// Mitsubishi GX Works2 project: BookEX6_54 Socket   PLC: Q13UDV

// global labels: Global
VAR_GLOBAL
  bVar0 AT M5000 : BOOL;
  abArray0 AT M5010 : ARRAY [0..49] OF BOOL;
  sStr0 AT D5000 : STRING[199];
  sStr1 AT D5100 : STRING[199];
  sStr2 AT D5200 : STRING[199];
  sStr3 AT D5300 : STRING[199];
  sStr4 AT D5400 : STRING[199];
  sStr5 AT D5500 : STRING[199];
  sStr6 AT D5600 : STRING[199];
  sStr7 AT D5700 : STRING[199];
  sStr8 AT D5800 : STRING[199];
  sStr9 AT D5900 : STRING[199];
  iVar0 AT D4500 : INT;
  iVar1 AT D4501 : INT;
  iVar2 AT D4502 : INT;
  iVar3 AT D4503 : INT;
  iVar4 AT D4504 : INT;
  iVar5 AT D4505 : INT;
  iVar6 AT D4506 : INT;
  iVar7 AT D4507 : INT;
  iVar8 AT D4508 : INT;
  iVar9 AT D4509 : INT;
  dVar0 AT D4510 : DINT;
  dVar1 AT D4512 : DINT;
  dVar2 AT D4514 : DINT;
  dVar3 AT D4516 : DINT;
  dVar4 AT D4518 : DINT;
  dVar5 AT D4520 : DINT;
  dVar6 AT D4522 : DINT;
  dVar7 AT D4524 : DINT;
  dVar8 AT D4526 : DINT;
  dVar9 AT D4528 : DINT;
  wVar0 AT D4530 : WORD;
  wVar1 AT D4531 : WORD;
  wVar2 AT D4532 : WORD;
  wVar3 AT D4533 : WORD;
  wVar4 AT D4534 : WORD;
  wVar5 AT D4535 : WORD;
  wVar6 AT D4536 : WORD;
  wVar7 AT D4537 : WORD;
  wVar8 AT D4538 : WORD;
  wVar9 AT D4539 : WORD;
  dwVar0 AT D4540 : DWORD;
  dwVar1 AT D4542 : DWORD;
  dwVar2 AT D4544 : DWORD;
  dwVar3 AT D4546 : DWORD;
  dwVar4 AT D4548 : DWORD;
  dwVar5 AT D4550 : DWORD;
  dwVar6 AT D4552 : DWORD;
  dwVar7 AT D4554 : DWORD;
  dwVar8 AT D4556 : DWORD;
  dwVar9 AT D4558 : DWORD;
  fsVar0 AT D4560 : REAL;
  fsVar1 AT D4562 : REAL;
  fsVar2 AT D4564 : REAL;
  fsVar3 AT D4566 : REAL;
  fsVar4 AT D4568 : REAL;
  fsVar5 AT D4570 : REAL;
  fsVar6 AT D4572 : REAL;
  fsVar7 AT D4574 : REAL;
  fsVar8 AT D4576 : REAL;
  fsVar9 AT D4578 : REAL;
  fdVar0 AT D4580 : LREAL;
  tTime0 AT D4620 : TIME;
  tTime1 AT D4622 : TIME;
  tTime2 AT D4624 : TIME;
  tTime3 AT D4626 : TIME;
  tTime4 AT D4628 : TIME;
  tTime5 AT D4630 : TIME;
  tTime6 AT D4632 : TIME;
  tTime7 AT D4634 : TIME;
  tTime8 AT D4636 : TIME;
  tTime9 AT D4638 : TIME;
  tTime10 AT D4640 : TIME;
  bVar1 AT M5001 : BOOL;
  bVar2 AT M5002 : BOOL;
  bVar3 AT M5003 : BOOL;
  bVar4 AT M5004 : BOOL;
  bVar5 AT M5005 : BOOL;
  bVar6 AT M5006 : BOOL;
  bVar7 AT M5007 : BOOL;
  bVar8 AT M5008 : BOOL;
  bVar9 AT M5009 : BOOL;
  abArray1 AT M5060 : ARRAY [0..49] OF BOOL;
  abArray2 AT M5110 : ARRAY [0..49] OF BOOL;
  abArray3 AT M5160 : ARRAY [0..49] OF BOOL;
  abArray4 AT M5210 : ARRAY [0..49] OF BOOL;
  abArray5 AT M5260 : ARRAY [0..49] OF BOOL;
  abArray6 AT M5310 : ARRAY [0..49] OF BOOL;
  abArray7 AT M5360 : ARRAY [0..49] OF BOOL;
  abArray8 AT M5410 : ARRAY [0..49] OF BOOL;
  abArray9 AT M5460 : ARRAY [0..49] OF BOOL;
  fdVar1 AT D4584 : LREAL;
  fdVar2 AT D4588 : LREAL;
  fdVar3 AT D4592 : LREAL;
  fdVar4 AT D4596 : LREAL;
  fdVar5 AT D4600 : LREAL;
  fdVar6 AT D4604 : LREAL;
  fdVar7 AT D4608 : LREAL;
  fdVar8 AT D4612 : LREAL;
  fdVar9 AT D4616 : LREAL;
END_VAR

// global labels: QPLCSpecial
VAR_GLOBAL
  sbGetTime AT SM213 : BOOL;
  sbOn AT SM400 : BOOL;
  sbOff AT SM401 : BOOL;
  sbOn1Time AT SM402 : BOOL;
  sbOff1Time AT SM403 : BOOL;
  sb5ms AT SM409 : BOOL;
  sdSwitch AT SD200 : INT;
  sdTime03 AT SD212 : INT;
  sdTime04 AT SD213 : INT;
  sdTime02 AT SD211 : INT;
  sdTime01 AT SD210 : INT;
  sdScanTime1 AT SD521 : INT;
  sdScanTimeMin1 AT SD525 : INT;
  sdScanTimeMin AT SD524 : INT;
  sdScanTimeMax1 AT SD527 : INT;
  sdScanTimeMax AT SD526 : INT;
  sbErrInfo2 AT SM16 : BOOL;
  sbErrInfo AT SM5 : BOOL;
  sbSelfError AT SM1 : BOOL;
  sbDiagError AT SM0 : BOOL;
  sbResetErr AT SM50 : BOOL;
  sbSetTime AT SM210 : BOOL;
  sbFuse AT SM60 : BOOL;
  sbOpError AT SM56 : BOOL;
  sbPowerDown AT SM53 : BOOL;
  sbBatLow AT SM52 : BOOL;
  sbBatLowL AT SM51 : BOOL;
  sbSTOP AT SM203 : BOOL;
  sbPAUSE AT SM204 : BOOL;
  sbNsec AT SM414 : BOOL;
  sb1000ms AT SM413 : BOOL;
  sb500ms AT SM412 : BOOL;
  sbNms AT SM415 : BOOL;
  sbUserClk4 AT SM424 : BOOL;
  sbUserClk3 AT SM423 : BOOL;
  sbUserClk2 AT SM422 : BOOL;
  sbUserClk1 AT SM421 : BOOL;
  sbUserClk0 AT SM420 : BOOL;
  sdBatLowL AT SD51 : INT;
  sdPLCErrInfo AT SD4 : INT;
  sdPLCErrDate2 AT SD3 : INT;
  sdPLCErrDate1 AT SD2 : INT;
  sdPLCErrDate0 AT SD1 : INT;
  sdPLCErrCode AT SD0 : INT;
  sdFuse AT SD60 : INT;
  sdPowerDown AT SD53 : INT;
  sdBatLow AT SD52 : INT;
  sdCPUSts AT SD203 : INT;
  sdLed AT SD201 : INT;
  sdScanTime AT SD520 : INT;
  sdCntNsec AT SD414 : INT;
  sdCnt1sec AT SD412 : INT;
  sdCntScan AT SD420 : INT;
  sdCntNms AT SD415 : INT;
  sb100ms AT SM411 : BOOL;
  sb50ms AT SM410 : BOOL;
  sdSckOpenComp AT SD1282 : WORD;
  sdSckOpenReq AT SD1284 : WORD;
  sdSckDataRx AT SD1286 : WORD;
  sdSckConn AT SD1288 : WORD;
END_VAR

// global labels: Network
VAR_GLOBAL
  aSendData1 AT D100 : ARRAY [0..4] OF INT;
  aiTxData AT D4000 : ARRAY [0..99] OF INT;
  aiRxData AT D4100 : ARRAY [0..99] OF INT;
  iOpenOK AT D3900 : INT;
  iOpenERR AT D3901 : INT;
  iSendOK AT D3902 : INT;
  iSendERR AT D3903 : INT;
  iCloseOK AT D3906 : INT;
  iCloseERR AT D3907 : INT;
  iRecvOK AT D3904 : INT;
  iRecvERR AT D3905 : INT;
  aiTxData2 AT D4200 : ARRAY [0..99] OF INT;
  aiRxData2 AT D4300 : ARRAY [0..99] OF INT;
  iOpenOK2 AT D3908 : INT;
  iOpenERR2 AT D3909 : INT;
  iSendOK2 AT D3910 : INT;
  iSendERR2 AT D3911 : INT;
  iRecvOK2 AT D3912 : INT;
  iRecvERR2 AT D3913 : INT;
  iCloseOK2 AT D3914 : INT;
  iCloseERR2 AT D3915 : INT;
  iEOpenComp AT D3916 : INT;
  iEOpenReq AT D3917 : INT;
  iERecvFlag AT D3918 : INT;
  iOpenCode AT D3919 : INT;
  iSendCode AT D3920 : INT;
  iRecvCode AT D3921 : INT;
  iCloseCode AT D3922 : INT;
  iOpenCode2 AT D3923 : INT;
  iSendCode2 AT D3924 : INT;
  iRecvCode2 AT D3925 : INT;
  iCloseCode2 AT D3926 : INT;
  aRecvData1 AT D105 : ARRAY [0..4] OF INT;
  aSendData2 AT D110 : ARRAY [0..4] OF INT;
  aRecvData2 AT D115 : ARRAY [0..4] OF INT;
  aSendData3 AT D120 : ARRAY [0..4] OF INT;
  aRecvData3 AT D125 : ARRAY [0..4] OF INT;
  aRdata AT D140 : ARRAY [0..9] OF INT;
  aSLMPDataTx AT D150 : ARRAY [0..9] OF WORD;
  aSLMPDataRx AT D160 : ARRAY [0..9] OF WORD;
END_VAR
// user libraries (not included): HMI

PROGRAM Ex_CactEpas
VAR
  bOpenReqC : BOOL;
  bOpenOkC : BOOL;
  bOpenErrC : BOOL;
  abOpenResC : ARRAY [0..1] OF BOOL;
  acOpenData : ARRAY [0..9] OF INT;
  bSendReqC : BOOL;
  bSendOkC : BOOL;
  bSendErrC : BOOL;
  abSendResC : ARRAY [0..1] OF BOOL;
  acSendDataC : ARRAY [0..1] OF INT;
  bRecvOkC : BOOL;
  bRecvErrC : BOOL;
  abRecvResC : ARRAY [0..1] OF BOOL;
  bCloseReq : BOOL;
  bCloseOkC : BOOL;
  bCloseErrC : BOOL;
  abCloseResC : ARRAY [0..1] OF BOOL;
  acCloseData : ARRAY [0..1] OF INT;
  CntSend1 : INT;
  CntSend2 : INT;
  CntRecv1 : INT;
  CntRecv2 : INT;
  Mov4INT_1 : Mov4INT;
  Mov8INT_1 : Mov8INT;
  acRdCtrl : ARRAY [0..9] OF INT;
  Mov4INT_2 : Mov4INT;
  bOpenReqE : BOOL;
  bOpenOkE : BOOL;
  bOpenErrE : BOOL;
  abOpenResE : ARRAY [0..1] OF BOOL;
  bSendErrE : BOOL;
  bSendOkE : BOOL;
  bSendReqE : BOOL;
  abSendResE : ARRAY [0..1] OF BOOL;
  abRecvResE : ARRAY [0..1] OF BOOL;
  bRecvErrE : BOOL;
  bRecvOkE : BOOL;
  abCloseResE : ARRAY [0..1] OF BOOL;
  bCloseErrE : BOOL;
  bCloseOkE : BOOL;
  acSendDataE : ARRAY [0..1] OF INT;
  acRecvDataC : ARRAY [0..1] OF INT;
  acRecvDataE : ARRAY [0..1] OF INT;
  Word2Bit8_1 : Word2Bit8;
  Word2Bit8_2 : Word2Bit8;
  Word2Bit8_3 : Word2Bit8;
  Word2Bit8_4 : Word2Bit8;
  Word2Bit8_5 : Word2Bit8;
  Word2Bit8_6 : Word2Bit8;
  ErrCodeSC : INT;
  ErrCodeSE : INT;
  Mov4INT_3 : Mov4INT;
  bChangeReqC : BOOL;
  Mov4INT_4 : Mov4INT;
  acRmodeData : ARRAY [0..3] OF INT;
  TON_1 : TON;
  CntRecvErr1 : INT;
  CntRecvErr2 : INT;
  TON_2 : TON;
  ErrCodeRC : INT;
  ErrCodeRE : INT;
  bModeReq : BOOL;
  acRdata : ARRAY [0..1] OF INT;
END_VAR
(* structured ladder/FBD written out as ST: instructions are called as NAME(EN, inputs, outputs); _pN, _eN, _tN stand for wires *)
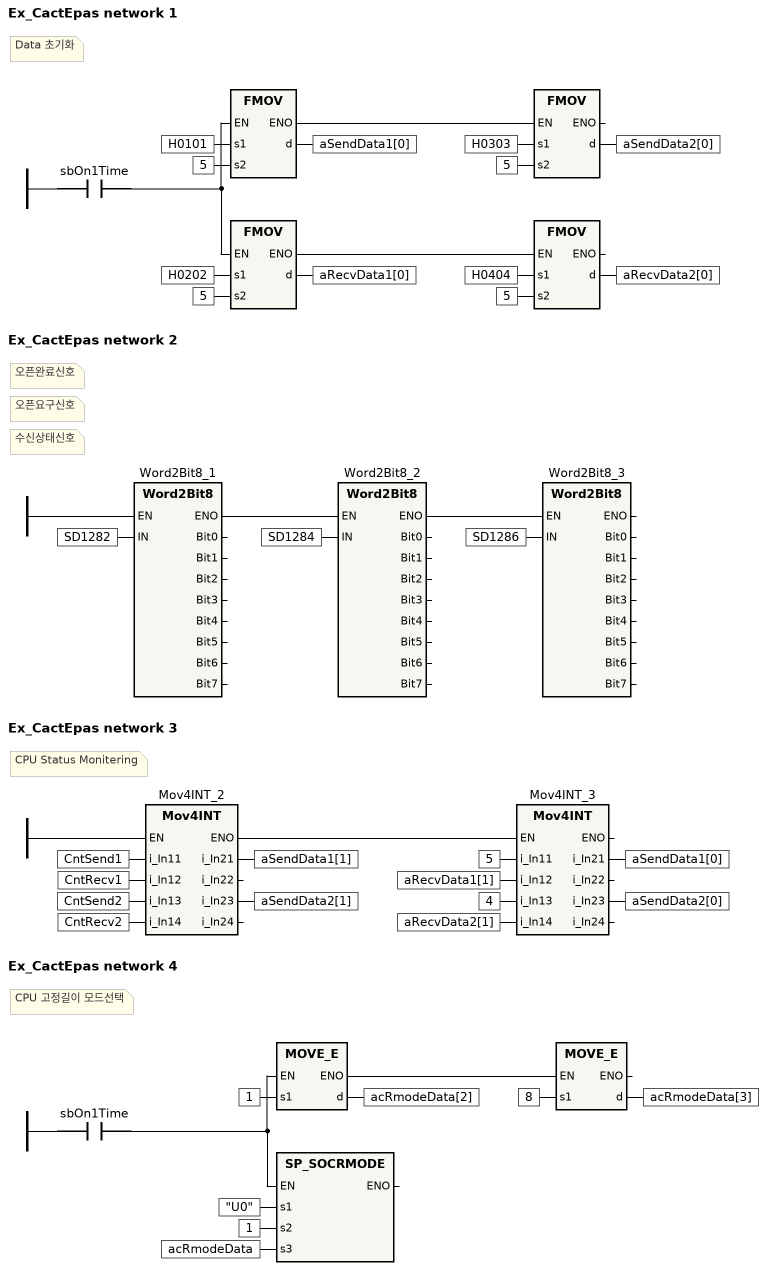
(* network 1 *)
(* Data 초기화 *)
_e1 := FMOV(sbOn1Time, H0101, 5, aSendData1[0]);
FMOV(_e1, H0303, 5, aSendData2[0]);
_e2 := FMOV(sbOn1Time, H0202, 5, aRecvData1[0]);
FMOV(_e2, H0404, 5, aRecvData2[0]);
(* network 2 *)
(* 오픈완료신호 *)
(* 오픈요구신호 *)
(* 수신상태신호 *)
Word2Bit8_1(EN := TRUE, IN := SD1282);
Word2Bit8_2(EN := Word2Bit8_1.ENO, IN := SD1284);
Word2Bit8_3(EN := Word2Bit8_2.ENO, IN := SD1286);
(* network 3 *)
(* CPU Status Monitering *)
Mov4INT_2(EN := TRUE, i_In11 := CntSend1, i_In12 := CntRecv1, i_In13 := CntSend2, i_In14 := CntRecv2, i_In21 => aSendData1[1], i_In23 => aSendData2[1]);
Mov4INT_3(EN := Mov4INT_2.ENO, i_In11 := 5, i_In12 := aRecvData1[1], i_In13 := 4, i_In14 := aRecvData2[1], i_In21 => aSendData1[0], i_In23 => aSendData2[0]);
(* network 4 *)
(* CPU 고정길이 모드선택 *)
_e1 := MOVE_E(sbOn1Time, 1, acRmodeData[2]);
MOVE_E(_e1, 8, acRmodeData[3]);
SP_SOCRMODE(sbOn1Time, "U0", 1, acRmodeData);
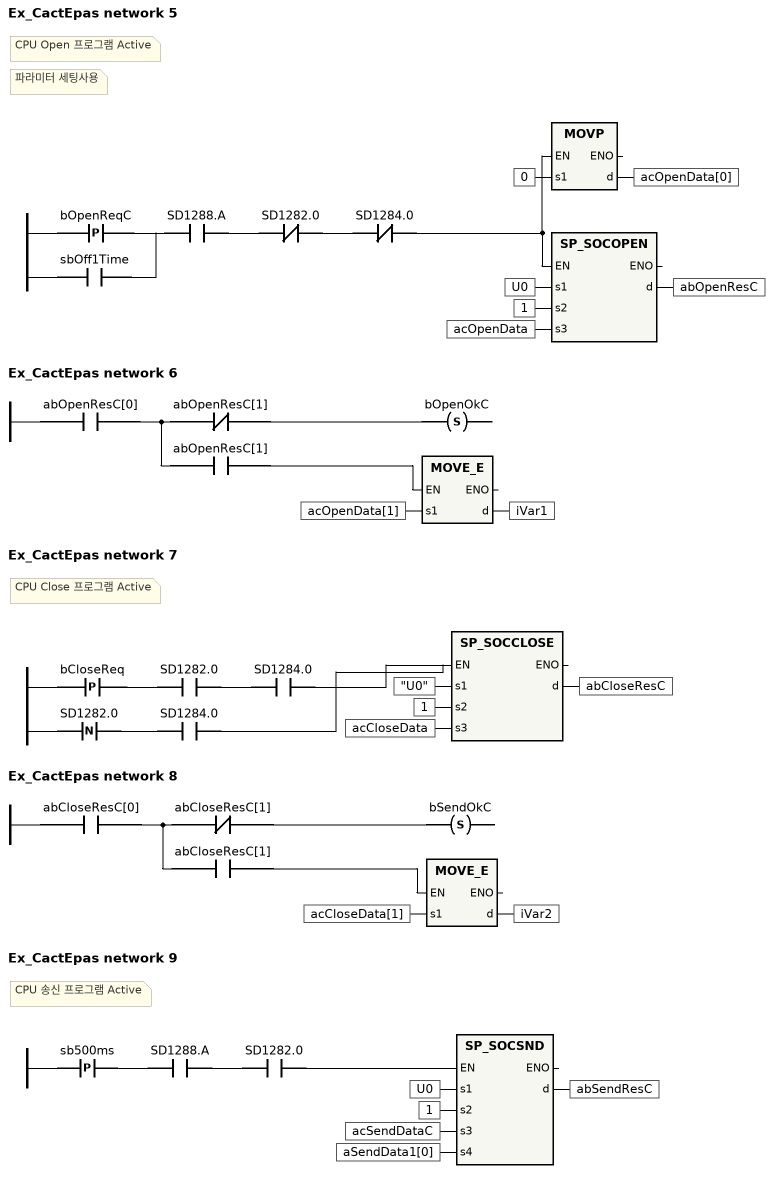
(* network 5 *)
(* CPU Open 프로그램 Active *)
(* 파라미터 세팅사용 *)
_p1 := (((LDP(TRUE, bOpenReqC) OR sbOff1Time) AND SD1288.A) AND NOT SD1282.0) AND NOT SD1284.0;
MOVP(_p1, 0, acOpenData[0]);
SP_SOCOPEN(_p1, U0, 1, acOpenData, abOpenResC);
(* network 6 *)
SET(abOpenResC[0] AND NOT abOpenResC[1], bOpenOkC);
MOVE_E(abOpenResC[0] AND abOpenResC[1], acOpenData[1], iVar1);
(* network 7 *)
(* CPU Close 프로그램 Active *)
SP_SOCCLOSE((LDP(TRUE, bCloseReq) AND SD1282.0 AND SD1284.0) OR (LDF(TRUE, SD1282.0) AND SD1284.0), "U0", 1, acCloseData, abCloseResC);
(* network 8 *)
SET(abCloseResC[0] AND NOT abCloseResC[1], bSendOkC);
MOVE_E(abCloseResC[0] AND abCloseResC[1], acCloseData[1], iVar2);
(* network 9 *)
(* CPU 송신 프로그램 Active *)
SP_SOCSND(LDP(TRUE, sb500ms) AND SD1288.A AND SD1282.0, U0, 1, acSendDataC, aSendData1[0], abSendResC);
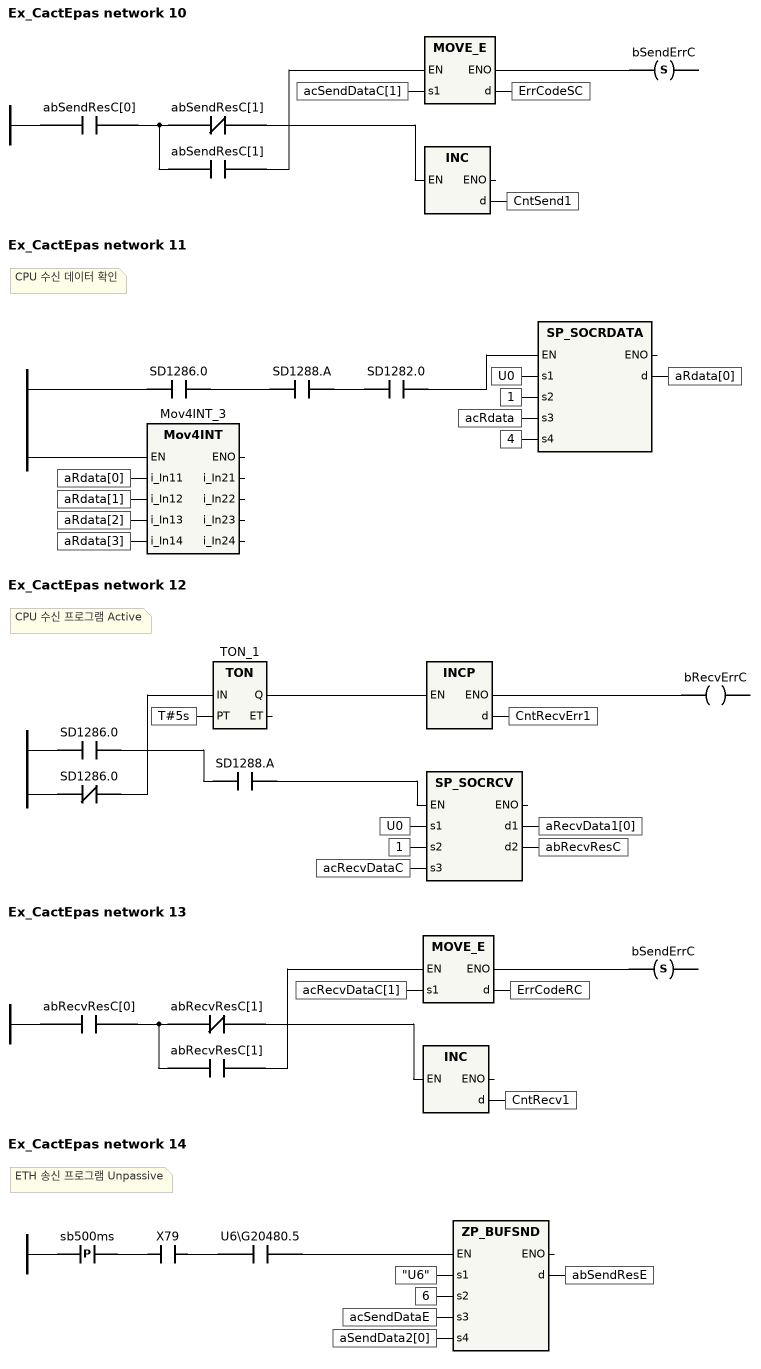
(* network 10 *)
INC(abSendResC[0] AND NOT abSendResC[1], CntSend1);
_e1 := MOVE_E(abSendResC[0] AND abSendResC[1], acSendDataC[1], ErrCodeSC);
SET(_e1, bSendErrC);
(* network 11 *)
(* CPU 수신 데이터 확인 *)
SP_SOCRDATA(SD1286.0 AND SD1288.A AND SD1282.0, U0, 1, acRdata, 4, aRdata[0]);
Mov4INT_3(EN := TRUE, i_In11 := aRdata[0], i_In12 := aRdata[1], i_In13 := aRdata[2], i_In14 := aRdata[3]);
(* network 12 *)
(* CPU 수신 프로그램 Active *)
SP_SOCRCV(SD1286.0 AND SD1288.A, U0, 1, acRecvDataC, aRecvData1[0], abRecvResC);
TON_1(IN := NOT SD1286.0, PT := T#5s);
_e1 := INCP(TON_1.Q, CntRecvErr1);
bRecvErrC := _e1;
(* network 13 *)
INC(abRecvResC[0] AND NOT abRecvResC[1], CntRecv1);
_e1 := MOVE_E(abRecvResC[0] AND abRecvResC[1], acRecvDataC[1], ErrCodeRC);
SET(_e1, bSendErrC);
(* network 14 *)
(* ETH 송신 프로그램 Unpassive *)
ZP_BUFSND(LDP(TRUE, sb500ms) AND X79 AND U6\G20480.5, "U6", 6, acSendDataE, aSendData2[0], abSendResE);
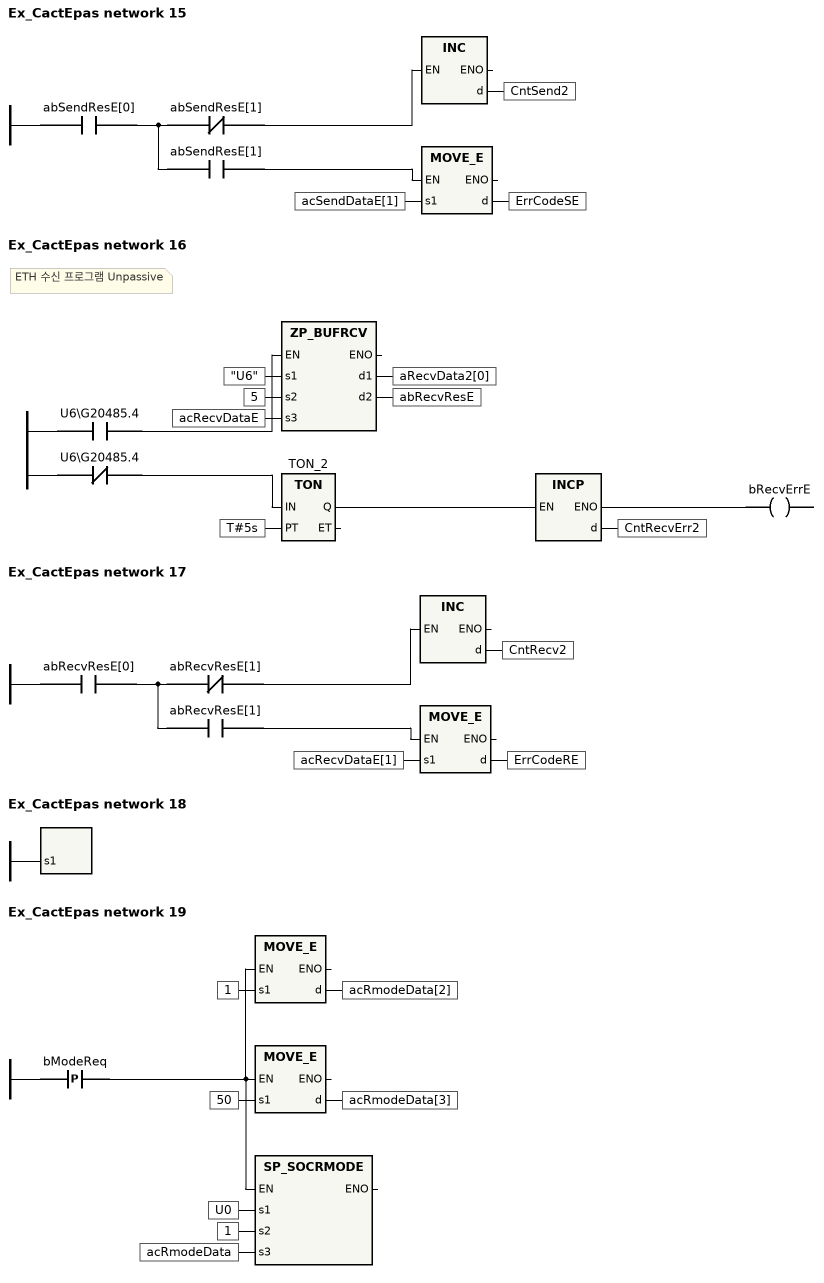
(* network 15 *)
INC(abSendResE[0] AND NOT abSendResE[1], CntSend2);
MOVE_E(abSendResE[0] AND abSendResE[1], acSendDataE[1], ErrCodeSE);
(* network 16 *)
(* ETH 수신 프로그램 Unpassive *)
ZP_BUFRCV(U6\G20485.4, "U6", 5, acRecvDataE, aRecvData2[0], abRecvResE);
TON_2(IN := NOT U6\G20485.4, PT := T#5s);
_e1 := INCP(TON_2.Q, CntRecvErr2);
bRecvErrE := _e1;
(* network 17 *)
INC(abRecvResE[0] AND NOT abRecvResE[1], CntRecv2);
MOVE_E(abRecvResE[0] AND abRecvResE[1], acRecvDataE[1], ErrCodeRE);
(* network 18 *)
(* element kind 10  <- TRUE *)
(* network 19 *)
_p1 := LDP(TRUE, bModeReq);
MOVE_E(_p1, 1, acRmodeData[2]);
MOVE_E(_p1, 50, acRmodeData[3]);
SP_SOCRMODE(_p1, U0, 1, acRmodeData);
END_PROGRAM

PROGRAM Ex_cpuREAD_WRITE
VAR
  Mov8INT_1 : Mov8INT;
  acRdCtrl : ARRAY [0..17] OF INT;
  abRdComp : ARRAY [0..1] OF BOOL;
  iCntRdOk : INT;
  iCntRdErr : INT;
END_VAR
(* structured ladder/FBD written out as ST: instructions are called as NAME(EN, inputs, outputs); _pN, _eN, _tN stand for wires *)
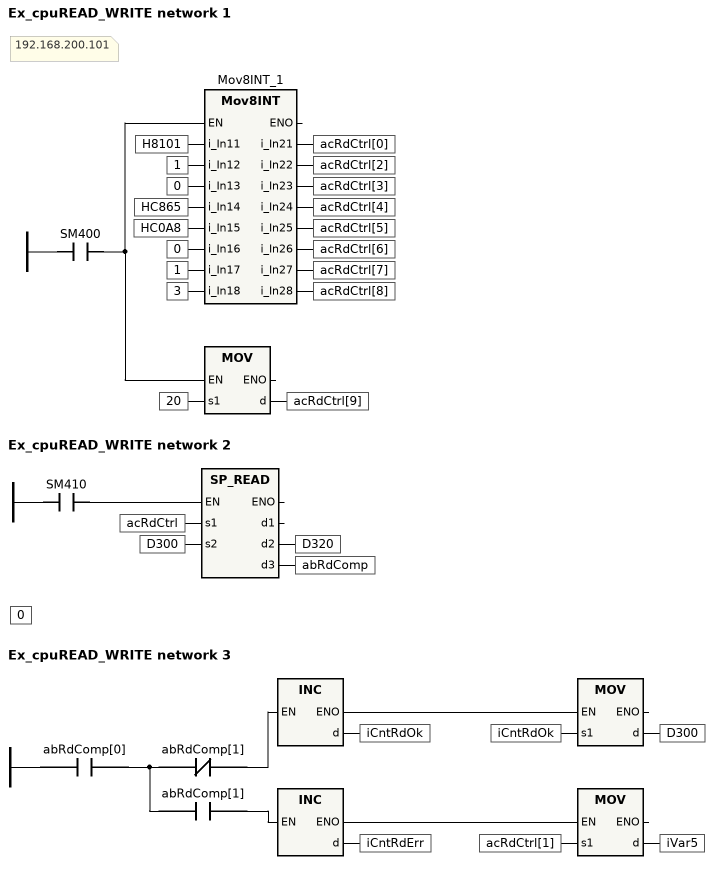
(* network 1 *)
(* 192.168.200.101 *)
Mov8INT_1(EN := SM400, i_In11 := H8101, i_In12 := 1, i_In13 := 0, i_In14 := HC865, i_In15 := HC0A8, i_In16 := 0, i_In17 := 1, i_In18 := 3, i_In21 => acRdCtrl[0], i_In22 => acRdCtrl[2], i_In23 => acRdCtrl[3], i_In24 => acRdCtrl[4], i_In25 => acRdCtrl[5], i_In26 => acRdCtrl[6], i_In27 => acRdCtrl[7], i_In28 => acRdCtrl[8]);
MOV(SM400, 20, acRdCtrl[9]);
(* network 2 *)
SP_READ(SM410, acRdCtrl, D300, _open, D320, abRdComp);
(* not connected to any output: 0 *)
(* network 3 *)
_e1 := INC(abRdComp[0] AND NOT abRdComp[1], iCntRdOk);
MOV(_e1, iCntRdOk, D300);
_e2 := INC(abRdComp[0] AND abRdComp[1], iCntRdErr);
MOV(_e2, acRdCtrl[1], iVar5);
END_PROGRAM

FUNCTION_BLOCK Word2Bit8
VAR_INPUT
  IN : WORD;
END_VAR
VAR_OUTPUT
  Bit0 : BOOL;
  Bit1 : BOOL;
  Bit2 : BOOL;
  Bit3 : BOOL;
  Bit4 : BOOL;
  Bit5 : BOOL;
  Bit6 : BOOL;
  Bit7 : BOOL;
END_VAR
 
Bit0 := WORD_TO_BOOL(IN AND 16#0001);
Bit1 := WORD_TO_BOOL(SHR(IN AND 16#0002 , 1));
Bit2 := WORD_TO_BOOL(SHR(IN AND 16#0004 , 2));
Bit3 := WORD_TO_BOOL(SHR(IN AND 16#0008 , 3));
Bit4 := WORD_TO_BOOL(SHR(IN AND 16#0010 , 4));
Bit5 := WORD_TO_BOOL(SHR(IN AND 16#0020 , 5));
Bit6 := WORD_TO_BOOL(SHR(IN AND 16#0040 , 6));
Bit7 := WORD_TO_BOOL(SHR(IN AND 16#0080 , 7));
END_FUNCTION_BLOCK

PROGRAM Ex_SOCCSET
VAR
  bOpenReqC : BOOL;
  bOpenOkC : BOOL;
  bOpenErrC : BOOL;
  abOpenResC : ARRAY [0..1] OF BOOL;
  acOpenData : ARRAY [0..9] OF INT;
  bSendReqC : BOOL;
  bSendOkC : BOOL;
  bSendErrC : BOOL;
  abSendResC : ARRAY [0..1] OF BOOL;
  acSendDataC : ARRAY [0..1] OF INT;
  bRecvOkC : BOOL;
  bRecvErrC : BOOL;
  abRecvResC : ARRAY [0..1] OF BOOL;
  bCloseReq : BOOL;
  bCloseOkC : BOOL;
  bCloseErrC : BOOL;
  abCloseResC : ARRAY [0..1] OF BOOL;
  acCloseData : ARRAY [0..1] OF INT;
  CntSend1 : INT;
  CntSend2 : INT;
  CntRecv1 : INT;
  CntRecv2 : INT;
  Mov4INT_1 : Mov4INT;
  Mov8INT_1 : Mov8INT;
  acRdCtrl : ARRAY [0..9] OF INT;
  Mov4INT_2 : Mov4INT;
  bOpenReqE : BOOL;
  bOpenOkE : BOOL;
  bOpenErrE : BOOL;
  abOpenResE : ARRAY [0..1] OF BOOL;
  bSendErrE : BOOL;
  bSendOkE : BOOL;
  bSendReqE : BOOL;
  abSendResE : ARRAY [0..1] OF BOOL;
  abRecvResE : ARRAY [0..1] OF BOOL;
  bRecvErrE : BOOL;
  bRecvOkE : BOOL;
  abCloseResE : ARRAY [0..1] OF BOOL;
  bCloseErrE : BOOL;
  bCloseOkE : BOOL;
  acSendDataE : ARRAY [0..1] OF INT;
  acRecvDataC : ARRAY [0..1] OF INT;
  acRecvDataE : ARRAY [0..1] OF INT;
  Word2Bit8_1 : Word2Bit8;
  Word2Bit8_2 : Word2Bit8;
  Word2Bit8_3 : Word2Bit8;
  Word2Bit8_4 : Word2Bit8;
  Word2Bit8_5 : Word2Bit8;
  Word2Bit8_6 : Word2Bit8;
  ErrCodeSC : INT;
  ErrCodeSE : INT;
  Mov4INT_3 : Mov4INT;
  bCsetReq : BOOL;
  Mov4INT_4 : Mov4INT;
  acCsetData : ARRAY [0..4] OF INT;
  TON_1 : TON;
  CntRecvErr1 : INT;
  CntRecvErr2 : INT;
  TON_2 : TON;
  ErrCodeRC : INT;
  ErrCodeRE : INT;
  CntSend3 : INT;
  CntRecv3 : INT;
  CntRecvErr3 : INT;
  abRecvResF : ARRAY [0..1] OF BOOL;
  acRecvDataF : ARRAY [0..1] OF INT;
  ErrCodeSF : INT;
  ErrCodeRF : INT;
  TON_3 : TON;
  bRecvErrF : BOOL;
  bRecvOkF : BOOL;
  acSendDataF : ARRAY [0..1] OF INT;
  abSendResF : ARRAY [0..1] OF BOOL;
END_VAR
(* structured ladder/FBD written out as ST: instructions are called as NAME(EN, inputs, outputs); _pN, _eN, _tN stand for wires *)
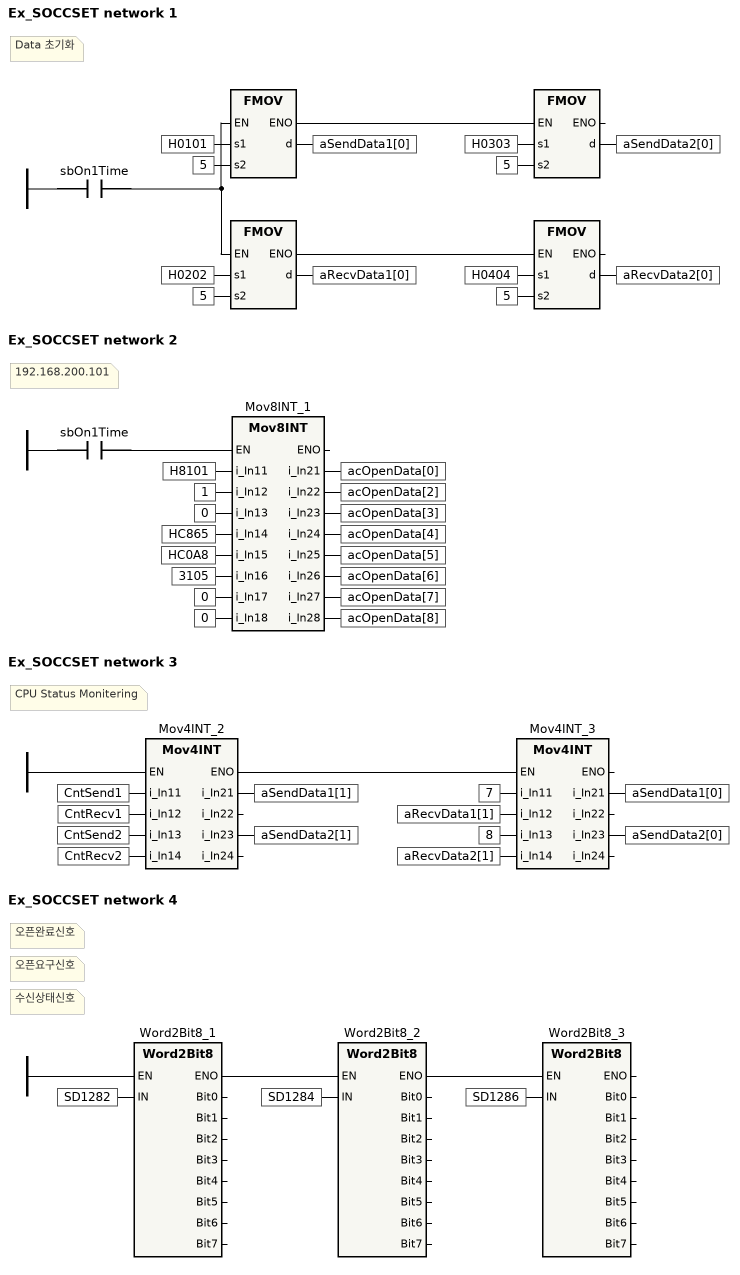
(* network 1 *)
(* Data 초기화 *)
_e1 := FMOV(sbOn1Time, H0101, 5, aSendData1[0]);
FMOV(_e1, H0303, 5, aSendData2[0]);
_e2 := FMOV(sbOn1Time, H0202, 5, aRecvData1[0]);
FMOV(_e2, H0404, 5, aRecvData2[0]);
(* network 2 *)
(* 192.168.200.101 *)
Mov8INT_1(EN := sbOn1Time, i_In11 := H8101, i_In12 := 1, i_In13 := 0, i_In14 := HC865, i_In15 := HC0A8, i_In16 := 3105, i_In17 := 0, i_In18 := 0, i_In21 => acOpenData[0], i_In22 => acOpenData[2], i_In23 => acOpenData[3], i_In24 => acOpenData[4], i_In25 => acOpenData[5], i_In26 => acOpenData[6], i_In27 => acOpenData[7], i_In28 => acOpenData[8]);
(* network 3 *)
(* CPU Status Monitering *)
Mov4INT_2(EN := TRUE, i_In11 := CntSend1, i_In12 := CntRecv1, i_In13 := CntSend2, i_In14 := CntRecv2, i_In21 => aSendData1[1], i_In23 => aSendData2[1]);
Mov4INT_3(EN := Mov4INT_2.ENO, i_In11 := 7, i_In12 := aRecvData1[1], i_In13 := 8, i_In14 := aRecvData2[1], i_In21 => aSendData1[0], i_In23 => aSendData2[0]);
(* network 4 *)
(* 오픈완료신호 *)
(* 오픈요구신호 *)
(* 수신상태신호 *)
Word2Bit8_1(EN := TRUE, IN := SD1282);
Word2Bit8_2(EN := Word2Bit8_1.ENO, IN := SD1284);
Word2Bit8_3(EN := Word2Bit8_2.ENO, IN := SD1286);
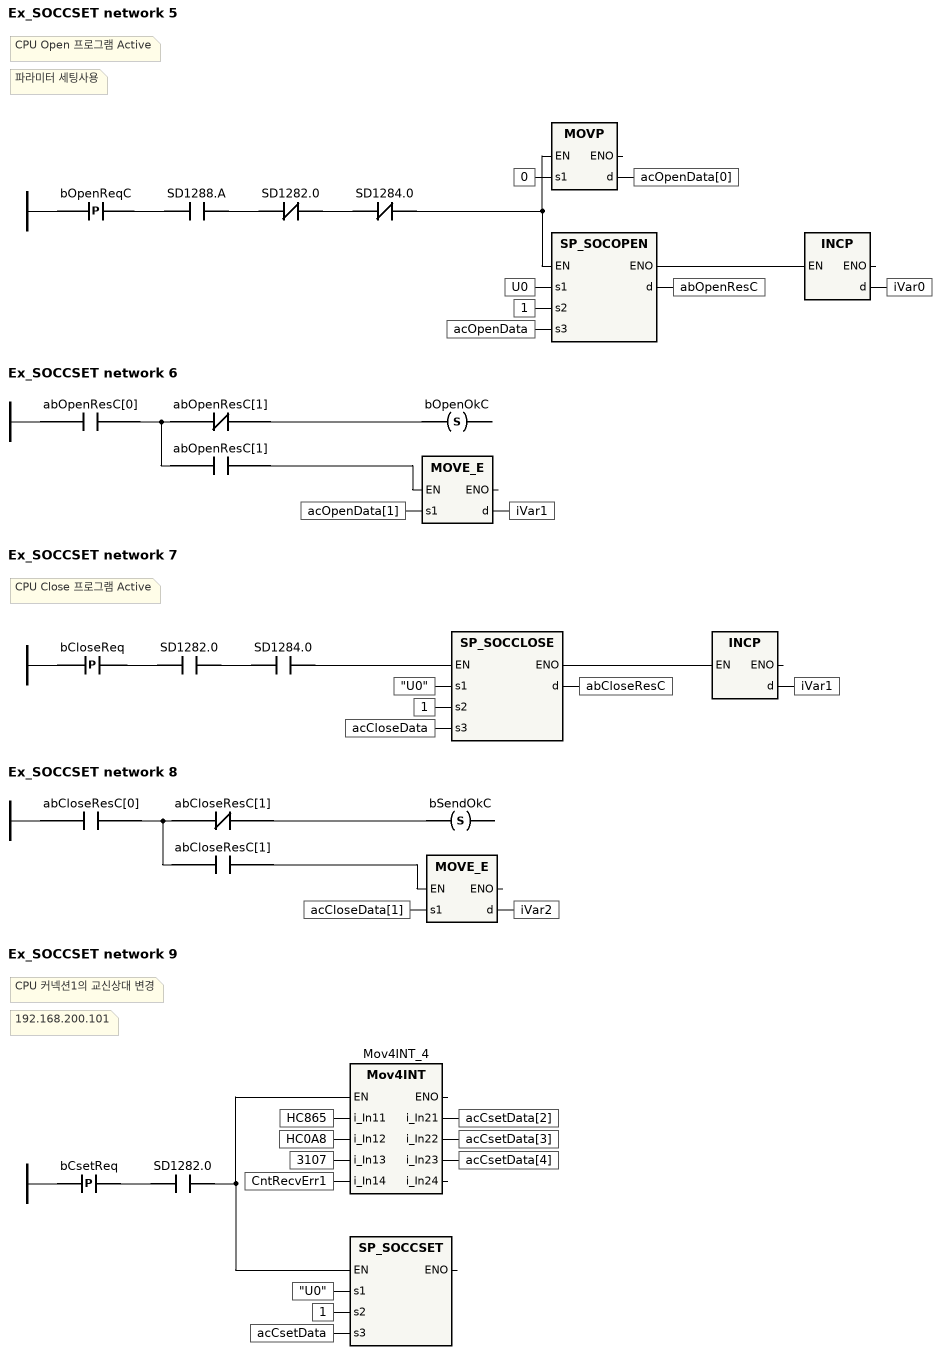
(* network 5 *)
(* CPU Open 프로그램 Active *)
(* 파라미터 세팅사용 *)
_p1 := LDP(TRUE, bOpenReqC) AND SD1288.A AND NOT SD1282.0 AND NOT SD1284.0;
MOVP(_p1, 0, acOpenData[0]);
_e2 := SP_SOCOPEN(_p1, U0, 1, acOpenData, abOpenResC);
INCP(_e2, iVar0);
(* network 6 *)
SET(abOpenResC[0] AND NOT abOpenResC[1], bOpenOkC);
MOVE_E(abOpenResC[0] AND abOpenResC[1], acOpenData[1], iVar1);
(* network 7 *)
(* CPU Close 프로그램 Active *)
_e1 := SP_SOCCLOSE(LDP(TRUE, bCloseReq) AND SD1282.0 AND SD1284.0, "U0", 1, acCloseData, abCloseResC);
INCP(_e1, iVar1);
(* network 8 *)
SET(abCloseResC[0] AND NOT abCloseResC[1], bSendOkC);
MOVE_E(abCloseResC[0] AND abCloseResC[1], acCloseData[1], iVar2);
(* network 9 *)
(* CPU 커넥션1의 교신상대 변경 *)
(* 192.168.200.101 *)
_p1 := LDP(TRUE, bCsetReq) AND SD1282.0;
Mov4INT_4(EN := _p1, i_In11 := HC865, i_In12 := HC0A8, i_In13 := 3107, i_In14 := CntRecvErr1, i_In21 => acCsetData[2], i_In22 => acCsetData[3], i_In23 => acCsetData[4]);
SP_SOCCSET(_p1, "U0", 1, acCsetData);
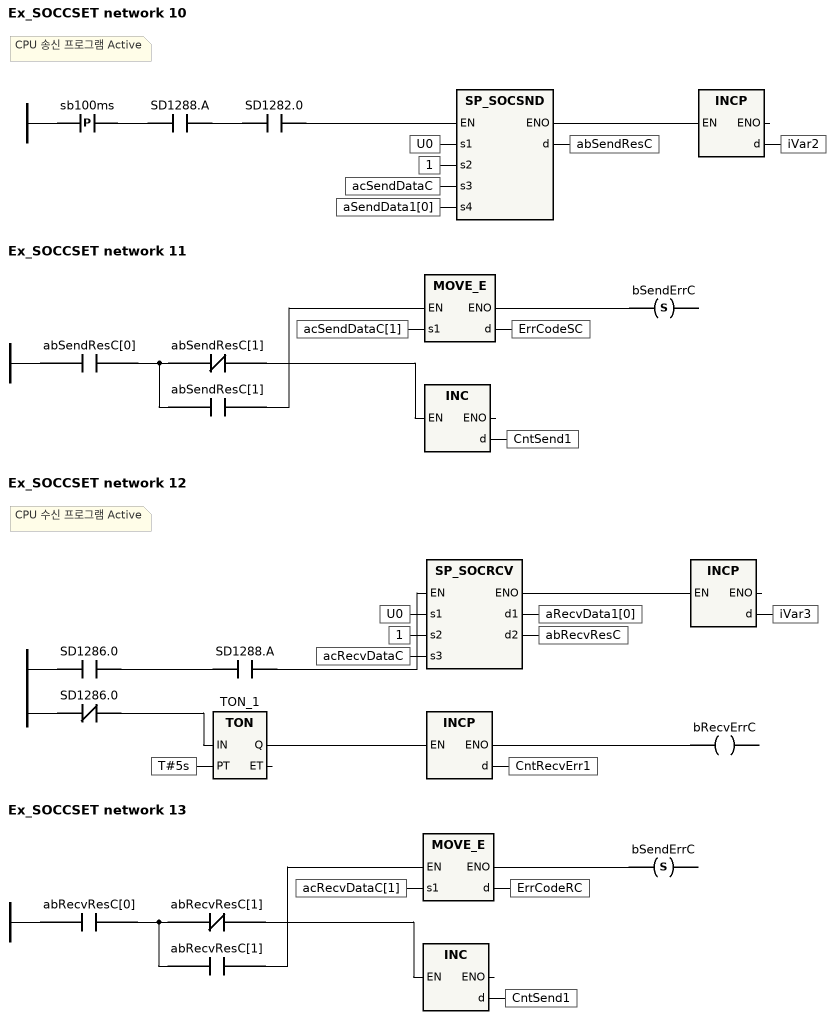
(* network 10 *)
(* CPU 송신 프로그램 Active *)
_e1 := SP_SOCSND(LDP(TRUE, sb100ms) AND SD1288.A AND SD1282.0, U0, 1, acSendDataC, aSendData1[0], abSendResC);
INCP(_e1, iVar2);
(* network 11 *)
INC(abSendResC[0] AND NOT abSendResC[1], CntSend1);
_e1 := MOVE_E(abSendResC[0] AND abSendResC[1], acSendDataC[1], ErrCodeSC);
SET(_e1, bSendErrC);
(* network 12 *)
(* CPU 수신 프로그램 Active *)
_e1 := SP_SOCRCV(SD1286.0 AND SD1288.A, U0, 1, acRecvDataC, aRecvData1[0], abRecvResC);
INCP(_e1, iVar3);
TON_1(IN := NOT SD1286.0, PT := T#5s);
_e2 := INCP(TON_1.Q, CntRecvErr1);
bRecvErrC := _e2;
(* network 13 *)
INC(abRecvResC[0] AND NOT abRecvResC[1], CntSend1);
_e1 := MOVE_E(abRecvResC[0] AND abRecvResC[1], acRecvDataC[1], ErrCodeRC);
SET(_e1, bSendErrC);
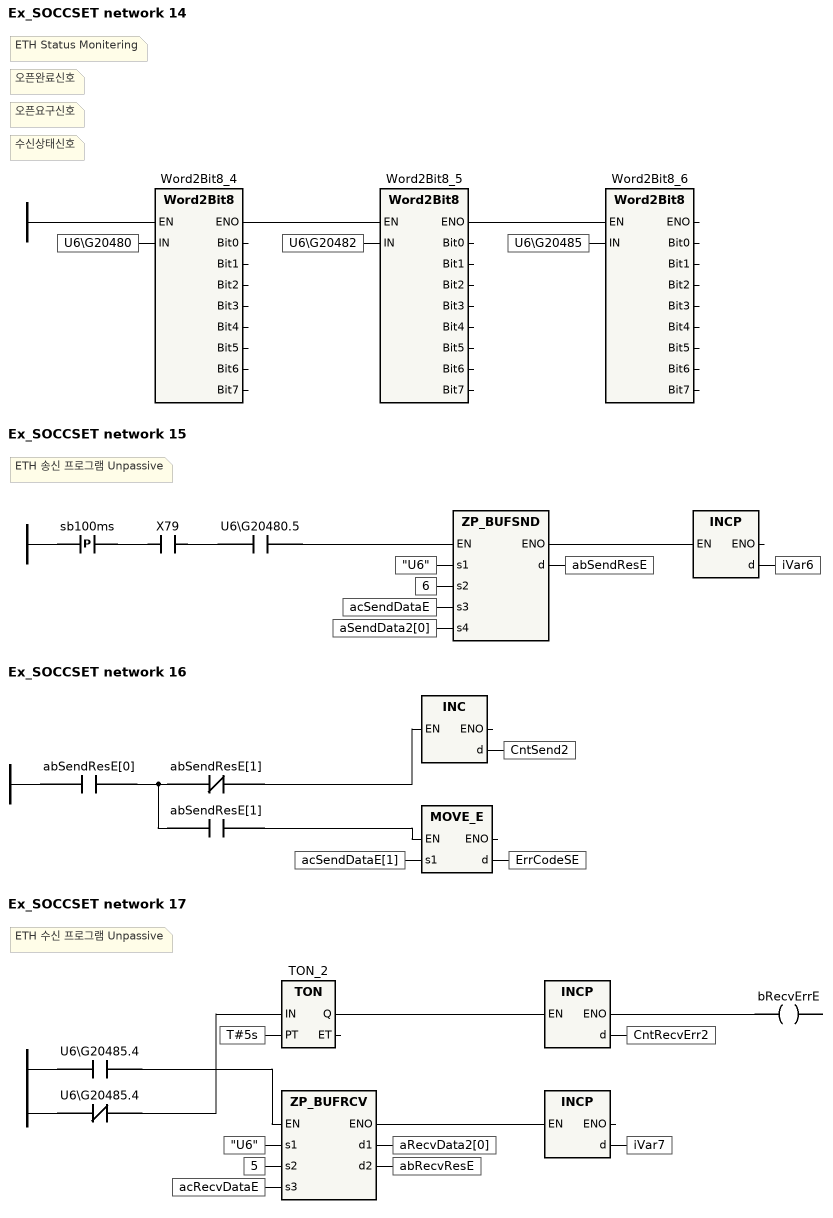
(* network 14 *)
(* ETH Status Monitering *)
(* 오픈완료신호 *)
(* 오픈요구신호 *)
(* 수신상태신호 *)
Word2Bit8_4(EN := TRUE, IN := U6\G20480);
Word2Bit8_5(EN := Word2Bit8_4.ENO, IN := U6\G20482);
Word2Bit8_6(EN := Word2Bit8_5.ENO, IN := U6\G20485);
(* network 15 *)
(* ETH 송신 프로그램 Unpassive *)
_e1 := ZP_BUFSND(LDP(TRUE, sb100ms) AND X79 AND U6\G20480.5, "U6", 6, acSendDataE, aSendData2[0], abSendResE);
INCP(_e1, iVar6);
(* network 16 *)
INC(abSendResE[0] AND NOT abSendResE[1], CntSend2);
MOVE_E(abSendResE[0] AND abSendResE[1], acSendDataE[1], ErrCodeSE);
(* network 17 *)
(* ETH 수신 프로그램 Unpassive *)
_e1 := ZP_BUFRCV(U6\G20485.4, "U6", 5, acRecvDataE, aRecvData2[0], abRecvResE);
INCP(_e1, iVar7);
TON_2(IN := NOT U6\G20485.4, PT := T#5s);
_e2 := INCP(TON_2.Q, CntRecvErr2);
bRecvErrE := _e2;
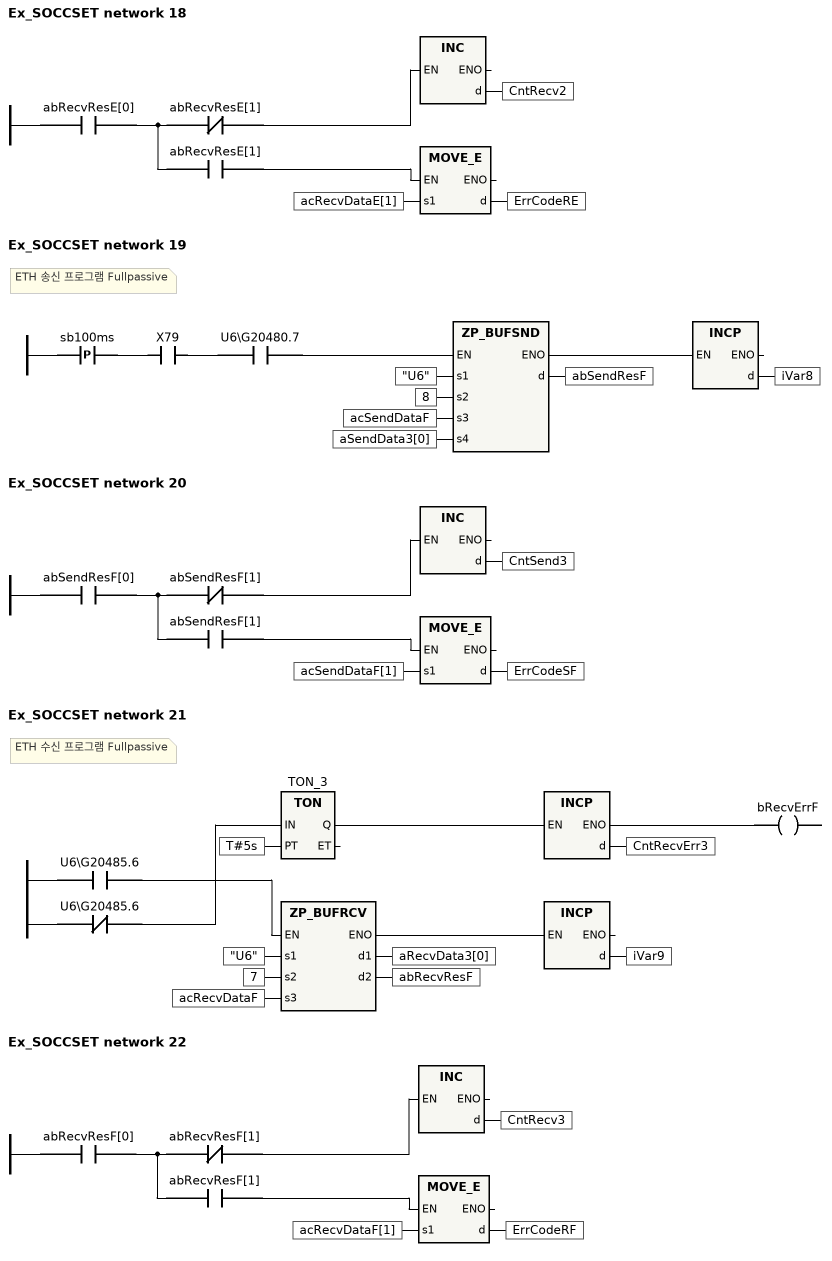
(* network 18 *)
INC(abRecvResE[0] AND NOT abRecvResE[1], CntRecv2);
MOVE_E(abRecvResE[0] AND abRecvResE[1], acRecvDataE[1], ErrCodeRE);
(* network 19 *)
(* ETH 송신 프로그램 Fullpassive *)
_e1 := ZP_BUFSND(LDP(TRUE, sb100ms) AND X79 AND U6\G20480.7, "U6", 8, acSendDataF, aSendData3[0], abSendResF);
INCP(_e1, iVar8);
(* network 20 *)
INC(abSendResF[0] AND NOT abSendResF[1], CntSend3);
MOVE_E(abSendResF[0] AND abSendResF[1], acSendDataF[1], ErrCodeSF);
(* network 21 *)
(* ETH 수신 프로그램 Fullpassive *)
_e1 := ZP_BUFRCV(U6\G20485.6, "U6", 7, acRecvDataF, aRecvData3[0], abRecvResF);
INCP(_e1, iVar9);
TON_3(IN := NOT U6\G20485.6, PT := T#5s);
_e2 := INCP(TON_3.Q, CntRecvErr3);
bRecvErrF := _e2;
(* network 22 *)
INC(abRecvResF[0] AND NOT abRecvResF[1], CntRecv3);
MOVE_E(abRecvResF[0] AND abRecvResF[1], acRecvDataF[1], ErrCodeRF);
END_PROGRAM

PROGRAM Ex_CactEfull
VAR
  bOpenReqC : BOOL;
  bCsetReq : BOOL;
  bOpenReqE : BOOL;
  bOpenOkC : BOOL;
  bOpenOkE : BOOL;
  bOpenErrC : BOOL;
  bOpenErrE : BOOL;
  abOpenResC : ARRAY [0..1] OF BOOL;
  abOpenResE : ARRAY [0..1] OF BOOL;
  acOpenData : ARRAY [0..9] OF INT;
  acCsetData : ARRAY [0..4] OF INT;
  acRdCtrl : ARRAY [0..9] OF INT;
  bSendReqC : BOOL;
  bSendReqE : BOOL;
  bSendOkC : BOOL;
  bSendOkE : BOOL;
  bSendErrC : BOOL;
  bSendErrE : BOOL;
  abSendResC : ARRAY [0..1] OF BOOL;
  abSendResE : ARRAY [0..1] OF BOOL;
  abSendResF : ARRAY [0..1] OF BOOL;
  acSendDataC : ARRAY [0..1] OF INT;
  acSendDataE : ARRAY [0..1] OF INT;
  acSendDataF : ARRAY [0..1] OF INT;
  bRecvOkC : BOOL;
  bRecvOkE : BOOL;
  bRecvOkF : BOOL;
  bRecvErrC : BOOL;
  bRecvErrE : BOOL;
  bRecvErrF : BOOL;
  abRecvResC : ARRAY [0..1] OF BOOL;
  abRecvResE : ARRAY [0..1] OF BOOL;
  abRecvResF : ARRAY [0..1] OF BOOL;
  acRecvDataC : ARRAY [0..1] OF INT;
  acRecvDataE : ARRAY [0..1] OF INT;
  acRecvDataF : ARRAY [0..1] OF INT;
  bCloseReq : BOOL;
  bCloseOkC : BOOL;
  bCloseOkE : BOOL;
  bCloseErrC : BOOL;
  bCloseErrE : BOOL;
  abCloseResC : ARRAY [0..1] OF BOOL;
  abCloseResE : ARRAY [0..1] OF BOOL;
  acCloseData : ARRAY [0..1] OF INT;
  CntSend1 : INT;
  CntSend2 : INT;
  CntSend3 : INT;
  CntRecv1 : INT;
  CntRecvErr1 : INT;
  CntRecv2 : INT;
  CntRecv3 : INT;
  CntRecvErr2 : INT;
  CntRecvErr3 : INT;
  ErrCodeSC : INT;
  ErrCodeSE : INT;
  ErrCodeSF : INT;
  ErrCodeRC : INT;
  ErrCodeRE : INT;
  ErrCodeRF : INT;
  Mov4INT_1 : Mov4INT;
  Mov8INT_1 : Mov8INT;
  Mov4INT_2 : Mov4INT;
  Mov4INT_3 : Mov4INT;
  Mov4INT_4 : Mov4INT;
  Word2Bit8_1 : Word2Bit8;
  Word2Bit8_2 : Word2Bit8;
  Word2Bit8_3 : Word2Bit8;
  Word2Bit8_4 : Word2Bit8;
  Word2Bit8_5 : Word2Bit8;
  Word2Bit8_6 : Word2Bit8;
  TON_1 : TON;
  TON_2 : TON;
  TON_3 : TON;
END_VAR
(* structured ladder/FBD written out as ST: instructions are called as NAME(EN, inputs, outputs); _pN, _eN, _tN stand for wires *)
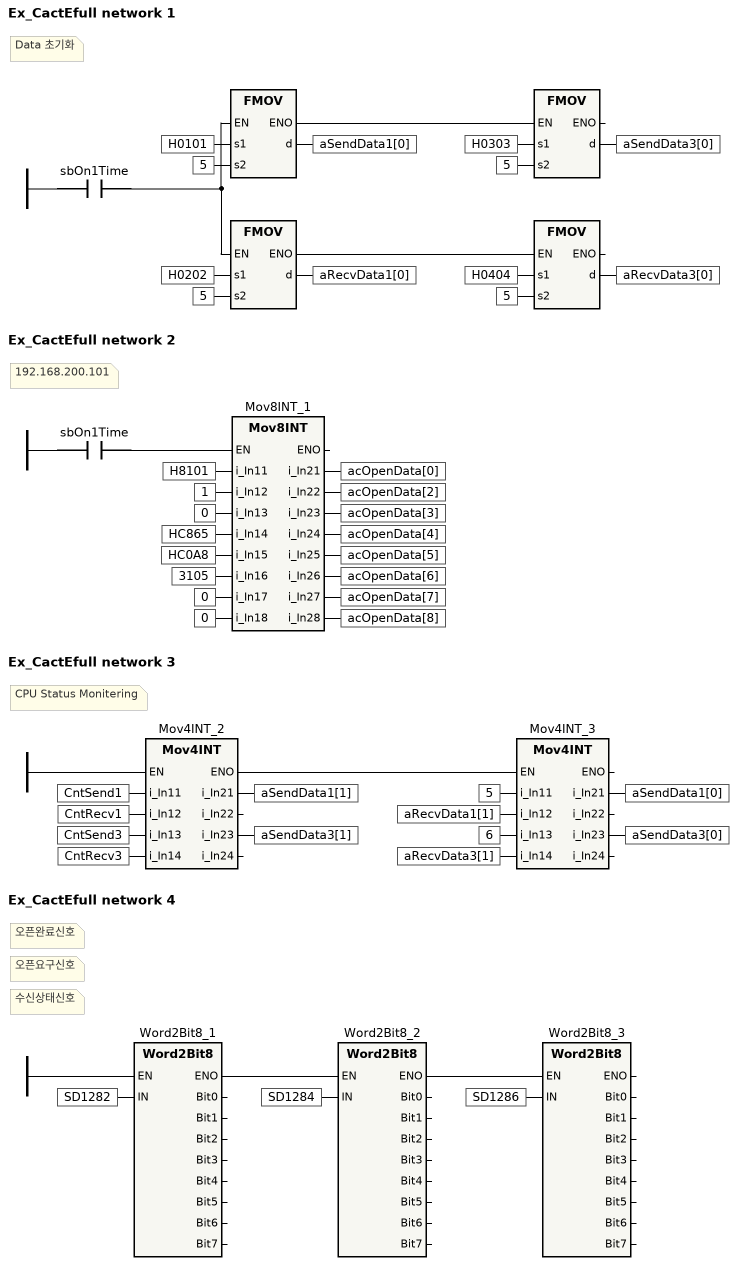
(* network 1 *)
(* Data 초기화 *)
_e1 := FMOV(sbOn1Time, H0101, 5, aSendData1[0]);
FMOV(_e1, H0303, 5, aSendData3[0]);
_e2 := FMOV(sbOn1Time, H0202, 5, aRecvData1[0]);
FMOV(_e2, H0404, 5, aRecvData3[0]);
(* network 2 *)
(* 192.168.200.101 *)
Mov8INT_1(EN := sbOn1Time, i_In11 := H8101, i_In12 := 1, i_In13 := 0, i_In14 := HC865, i_In15 := HC0A8, i_In16 := 3105, i_In17 := 0, i_In18 := 0, i_In21 => acOpenData[0], i_In22 => acOpenData[2], i_In23 => acOpenData[3], i_In24 => acOpenData[4], i_In25 => acOpenData[5], i_In26 => acOpenData[6], i_In27 => acOpenData[7], i_In28 => acOpenData[8]);
(* network 3 *)
(* CPU Status Monitering *)
Mov4INT_2(EN := TRUE, i_In11 := CntSend1, i_In12 := CntRecv1, i_In13 := CntSend3, i_In14 := CntRecv3, i_In21 => aSendData1[1], i_In23 => aSendData3[1]);
Mov4INT_3(EN := Mov4INT_2.ENO, i_In11 := 5, i_In12 := aRecvData1[1], i_In13 := 6, i_In14 := aRecvData3[1], i_In21 => aSendData1[0], i_In23 => aSendData3[0]);
(* network 4 *)
(* 오픈완료신호 *)
(* 오픈요구신호 *)
(* 수신상태신호 *)
Word2Bit8_1(EN := TRUE, IN := SD1282);
Word2Bit8_2(EN := Word2Bit8_1.ENO, IN := SD1284);
Word2Bit8_3(EN := Word2Bit8_2.ENO, IN := SD1286);
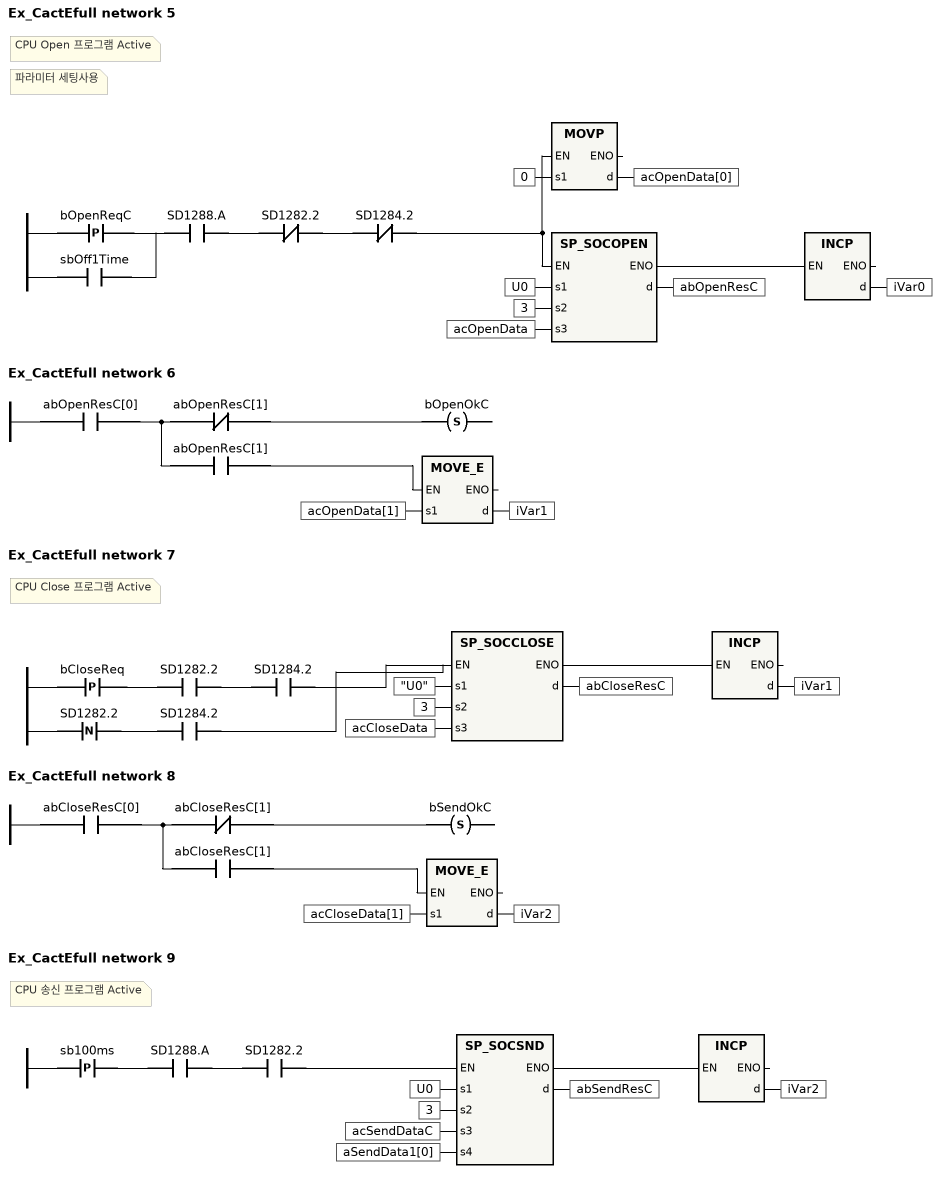
(* network 5 *)
(* CPU Open 프로그램 Active *)
(* 파라미터 세팅사용 *)
_p1 := (((LDP(TRUE, bOpenReqC) OR sbOff1Time) AND SD1288.A) AND NOT SD1282.2) AND NOT SD1284.2;
MOVP(_p1, 0, acOpenData[0]);
_e2 := SP_SOCOPEN(_p1, U0, 3, acOpenData, abOpenResC);
INCP(_e2, iVar0);
(* network 6 *)
SET(abOpenResC[0] AND NOT abOpenResC[1], bOpenOkC);
MOVE_E(abOpenResC[0] AND abOpenResC[1], acOpenData[1], iVar1);
(* network 7 *)
(* CPU Close 프로그램 Active *)
_e1 := SP_SOCCLOSE((LDP(TRUE, bCloseReq) AND SD1282.2 AND SD1284.2) OR (LDF(TRUE, SD1282.2) AND SD1284.2), "U0", 3, acCloseData, abCloseResC);
INCP(_e1, iVar1);
(* network 8 *)
SET(abCloseResC[0] AND NOT abCloseResC[1], bSendOkC);
MOVE_E(abCloseResC[0] AND abCloseResC[1], acCloseData[1], iVar2);
(* network 9 *)
(* CPU 송신 프로그램 Active *)
_e1 := SP_SOCSND(LDP(TRUE, sb100ms) AND SD1288.A AND SD1282.2, U0, 3, acSendDataC, aSendData1[0], abSendResC);
INCP(_e1, iVar2);
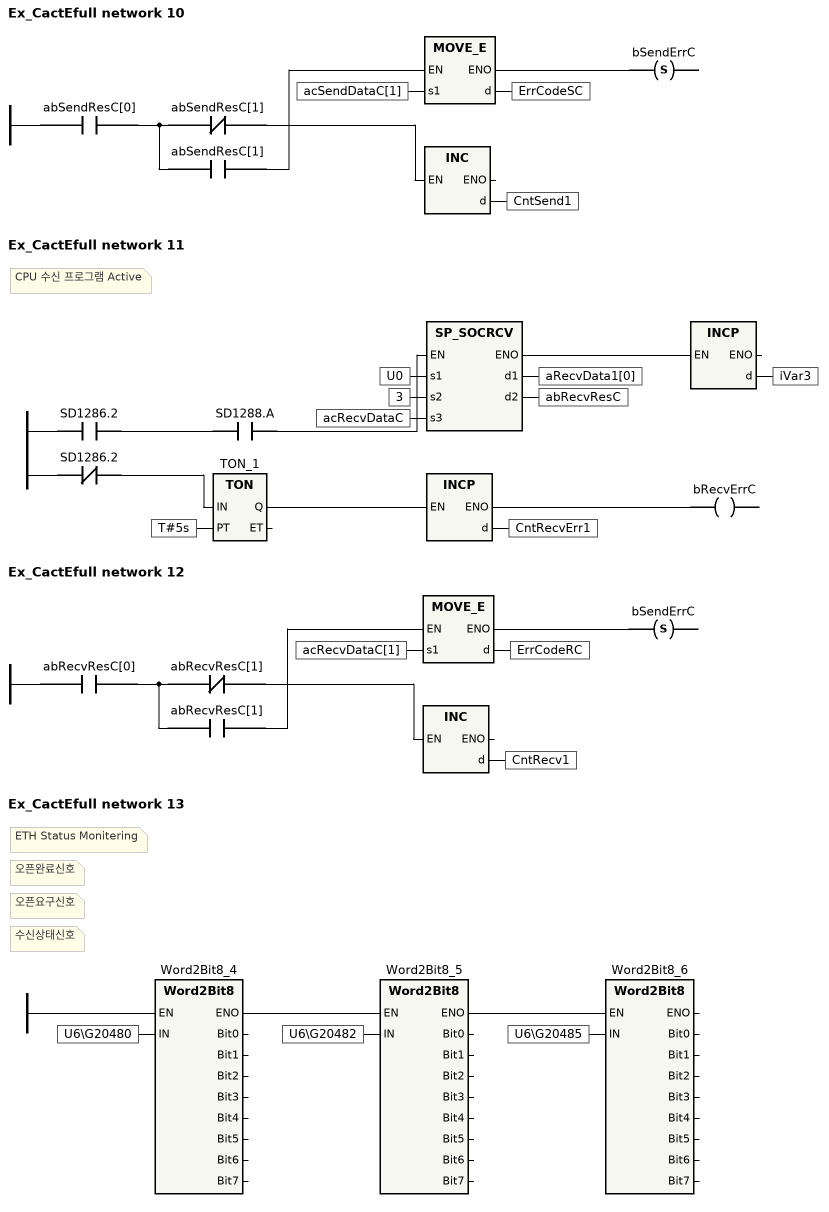
(* network 10 *)
INC(abSendResC[0] AND NOT abSendResC[1], CntSend1);
_e1 := MOVE_E(abSendResC[0] AND abSendResC[1], acSendDataC[1], ErrCodeSC);
SET(_e1, bSendErrC);
(* network 11 *)
(* CPU 수신 프로그램 Active *)
_e1 := SP_SOCRCV(SD1286.2 AND SD1288.A, U0, 3, acRecvDataC, aRecvData1[0], abRecvResC);
INCP(_e1, iVar3);
TON_1(IN := NOT SD1286.2, PT := T#5s);
_e2 := INCP(TON_1.Q, CntRecvErr1);
bRecvErrC := _e2;
(* network 12 *)
INC(abRecvResC[0] AND NOT abRecvResC[1], CntRecv1);
_e1 := MOVE_E(abRecvResC[0] AND abRecvResC[1], acRecvDataC[1], ErrCodeRC);
SET(_e1, bSendErrC);
(* network 13 *)
(* ETH Status Monitering *)
(* 오픈완료신호 *)
(* 오픈요구신호 *)
(* 수신상태신호 *)
Word2Bit8_4(EN := TRUE, IN := U6\G20480);
Word2Bit8_5(EN := Word2Bit8_4.ENO, IN := U6\G20482);
Word2Bit8_6(EN := Word2Bit8_5.ENO, IN := U6\G20485);
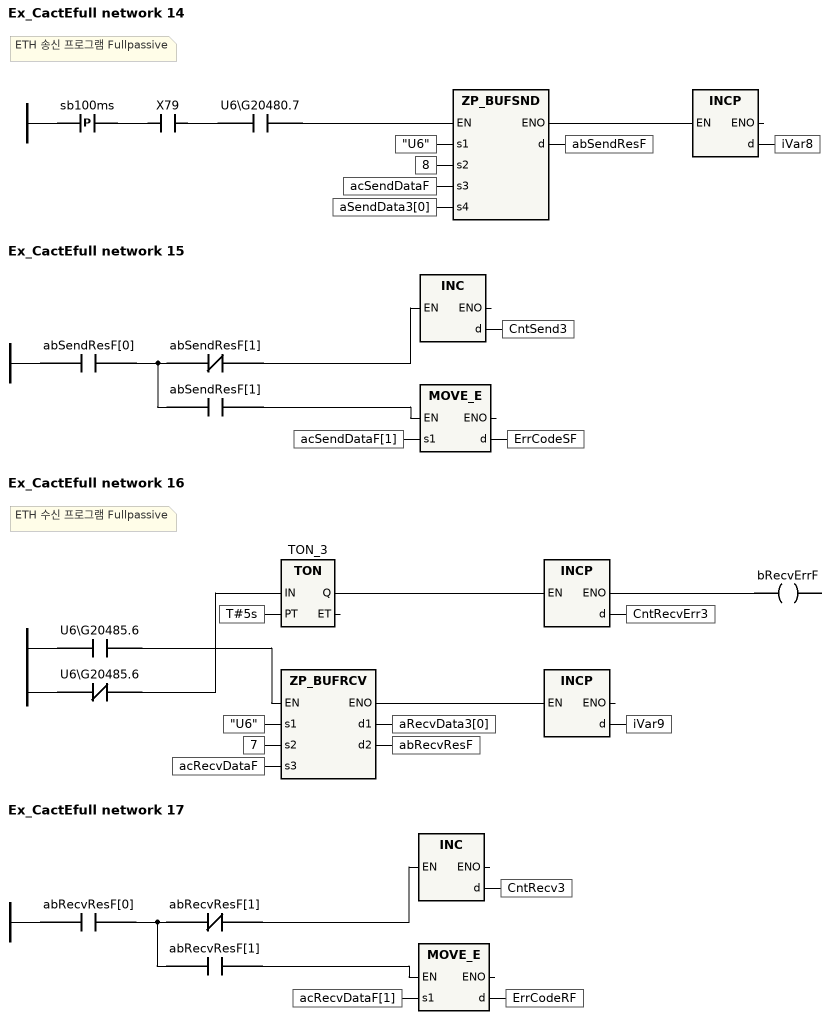
(* network 14 *)
(* ETH 송신 프로그램 Fullpassive *)
_e1 := ZP_BUFSND(LDP(TRUE, sb100ms) AND X79 AND U6\G20480.7, "U6", 8, acSendDataF, aSendData3[0], abSendResF);
INCP(_e1, iVar8);
(* network 15 *)
INC(abSendResF[0] AND NOT abSendResF[1], CntSend3);
MOVE_E(abSendResF[0] AND abSendResF[1], acSendDataF[1], ErrCodeSF);
(* network 16 *)
(* ETH 수신 프로그램 Fullpassive *)
_e1 := ZP_BUFRCV(U6\G20485.6, "U6", 7, acRecvDataF, aRecvData3[0], abRecvResF);
INCP(_e1, iVar9);
TON_3(IN := NOT U6\G20485.6, PT := T#5s);
_e2 := INCP(TON_3.Q, CntRecvErr3);
bRecvErrF := _e2;
(* network 17 *)
INC(abRecvResF[0] AND NOT abRecvResF[1], CntRecv3);
MOVE_E(abRecvResF[0] AND abRecvResF[1], acRecvDataF[1], ErrCodeRF);
END_PROGRAM

PROGRAM Ex_CactFact
VAR
  bOpenReqC : BOOL;
  bOpenOkC : BOOL;
  bOpenErrC : BOOL;
  abOpenResC : ARRAY [0..1] OF BOOL;
  acOpenDataC : ARRAY [0..9] OF INT;
  bSendReqC : BOOL;
  bSendOkC : BOOL;
  bSendErrC : BOOL;
  abSendResC : ARRAY [0..1] OF BOOL;
  acSendDataC : ARRAY [0..1] OF INT;
  bRecvOkC : BOOL;
  bRecvErrC : BOOL;
  abRecvResC : ARRAY [0..1] OF BOOL;
  bCloseReqC : BOOL;
  bCloseOkC : BOOL;
  bCloseErrC : BOOL;
  abCloseResC : ARRAY [0..1] OF BOOL;
  acCloseDataC : ARRAY [0..1] OF INT;
  CntSend1 : INT;
  CntSend2 : INT;
  CntRecv1 : INT;
  CntRecv2 : INT;
  Mov4INT_1 : Mov4INT;
  Mov8INT_1 : Mov8INT;
  acRdCtrl : ARRAY [0..9] OF INT;
  Mov4INT_2 : Mov4INT;
  bOpenReqE : BOOL;
  bOpenOkE : BOOL;
  bOpenErrE : BOOL;
  abOpenResE : ARRAY [0..1] OF BOOL;
  bSendErrE : BOOL;
  bSendOkE : BOOL;
  bSendReqE : BOOL;
  abSendResE : ARRAY [0..1] OF BOOL;
  abRecvResE : ARRAY [0..1] OF BOOL;
  bRecvErrE : BOOL;
  bRecvOkE : BOOL;
  abCloseResE : ARRAY [0..1] OF BOOL;
  bCloseErrE : BOOL;
  bCloseOkE : BOOL;
  acSendDataE : ARRAY [0..1] OF INT;
  acRecvDataC : ARRAY [0..1] OF INT;
  acRecvDataE : ARRAY [0..1] OF INT;
  Word2Bit8_1 : Word2Bit8;
  Word2Bit8_2 : Word2Bit8;
  Word2Bit8_3 : Word2Bit8;
  Word2Bit8_4 : Word2Bit8;
  Word2Bit8_5 : Word2Bit8;
  Word2Bit8_6 : Word2Bit8;
  ErrCodeSC : INT;
  ErrCodeSE : INT;
  Mov4INT_3 : Mov4INT;
  bChangeReqC : BOOL;
  Mov4INT_4 : Mov4INT;
  acCsetData : ARRAY [0..4] OF INT;
  TON_1 : TON;
  CntRecvErr1 : INT;
  CntRecvErr2 : INT;
  TON_2 : TON;
  ErrCodeRC : INT;
  ErrCodeRE : INT;
  bCloseReqE : BOOL;
  acOpenDataE : ARRAY [0..9] OF INT;
  acCloseDataE : ARRAY [0..1] OF INT;
END_VAR
(* structured ladder/FBD written out as ST: instructions are called as NAME(EN, inputs, outputs); _pN, _eN, _tN stand for wires *)
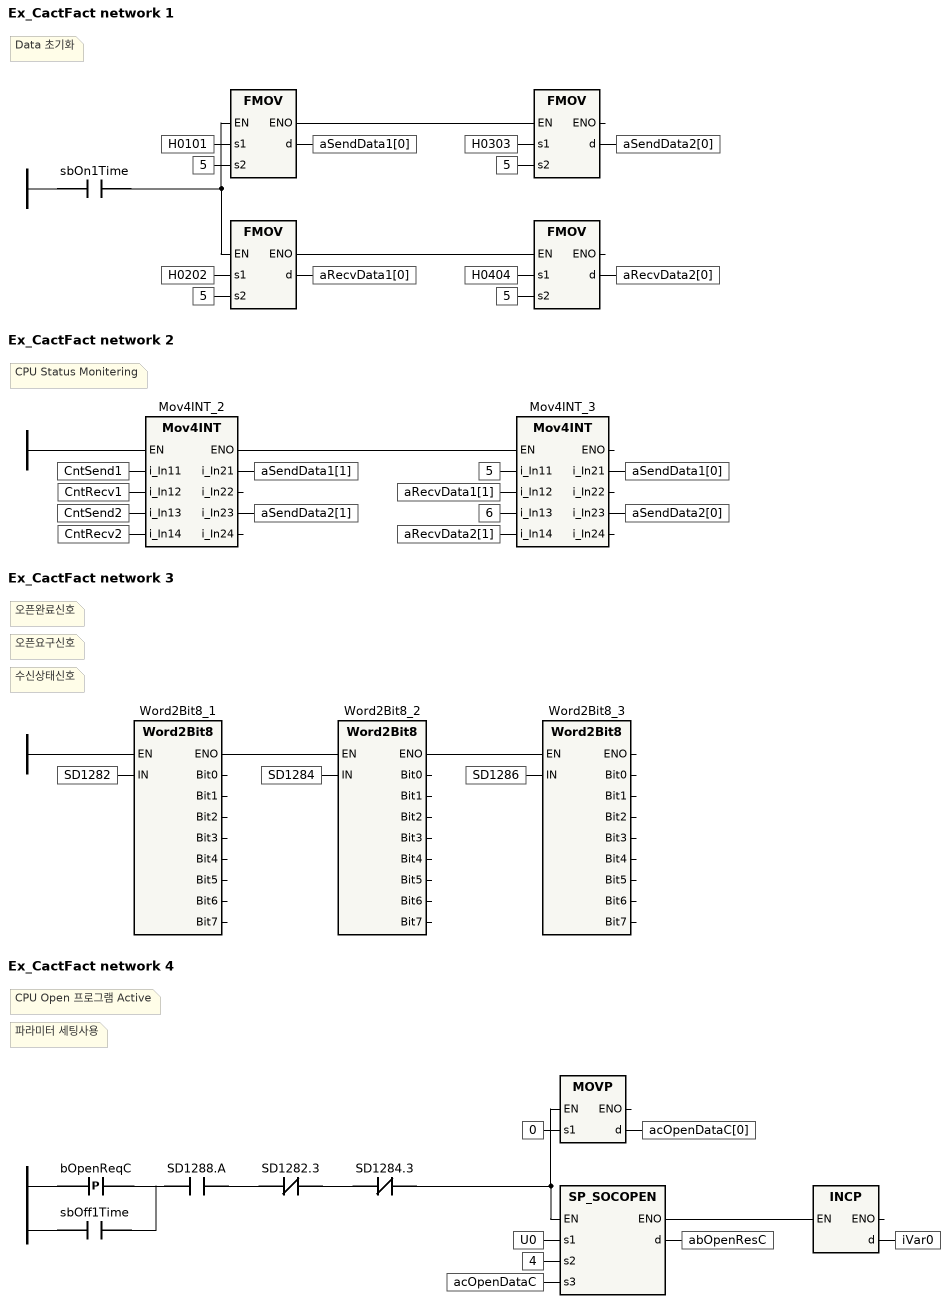
(* network 1 *)
(* Data 초기화 *)
_e1 := FMOV(sbOn1Time, H0101, 5, aSendData1[0]);
FMOV(_e1, H0303, 5, aSendData2[0]);
_e2 := FMOV(sbOn1Time, H0202, 5, aRecvData1[0]);
FMOV(_e2, H0404, 5, aRecvData2[0]);
(* network 2 *)
(* CPU Status Monitering *)
Mov4INT_2(EN := TRUE, i_In11 := CntSend1, i_In12 := CntRecv1, i_In13 := CntSend2, i_In14 := CntRecv2, i_In21 => aSendData1[1], i_In23 => aSendData2[1]);
Mov4INT_3(EN := Mov4INT_2.ENO, i_In11 := 5, i_In12 := aRecvData1[1], i_In13 := 6, i_In14 := aRecvData2[1], i_In21 => aSendData1[0], i_In23 => aSendData2[0]);
(* network 3 *)
(* 오픈완료신호 *)
(* 오픈요구신호 *)
(* 수신상태신호 *)
Word2Bit8_1(EN := TRUE, IN := SD1282);
Word2Bit8_2(EN := Word2Bit8_1.ENO, IN := SD1284);
Word2Bit8_3(EN := Word2Bit8_2.ENO, IN := SD1286);
(* network 4 *)
(* CPU Open 프로그램 Active *)
(* 파라미터 세팅사용 *)
_p1 := (((LDP(TRUE, bOpenReqC) OR sbOff1Time) AND SD1288.A) AND NOT SD1282.3) AND NOT SD1284.3;
MOVP(_p1, 0, acOpenDataC[0]);
_e2 := SP_SOCOPEN(_p1, U0, 4, acOpenDataC, abOpenResC);
INCP(_e2, iVar0);
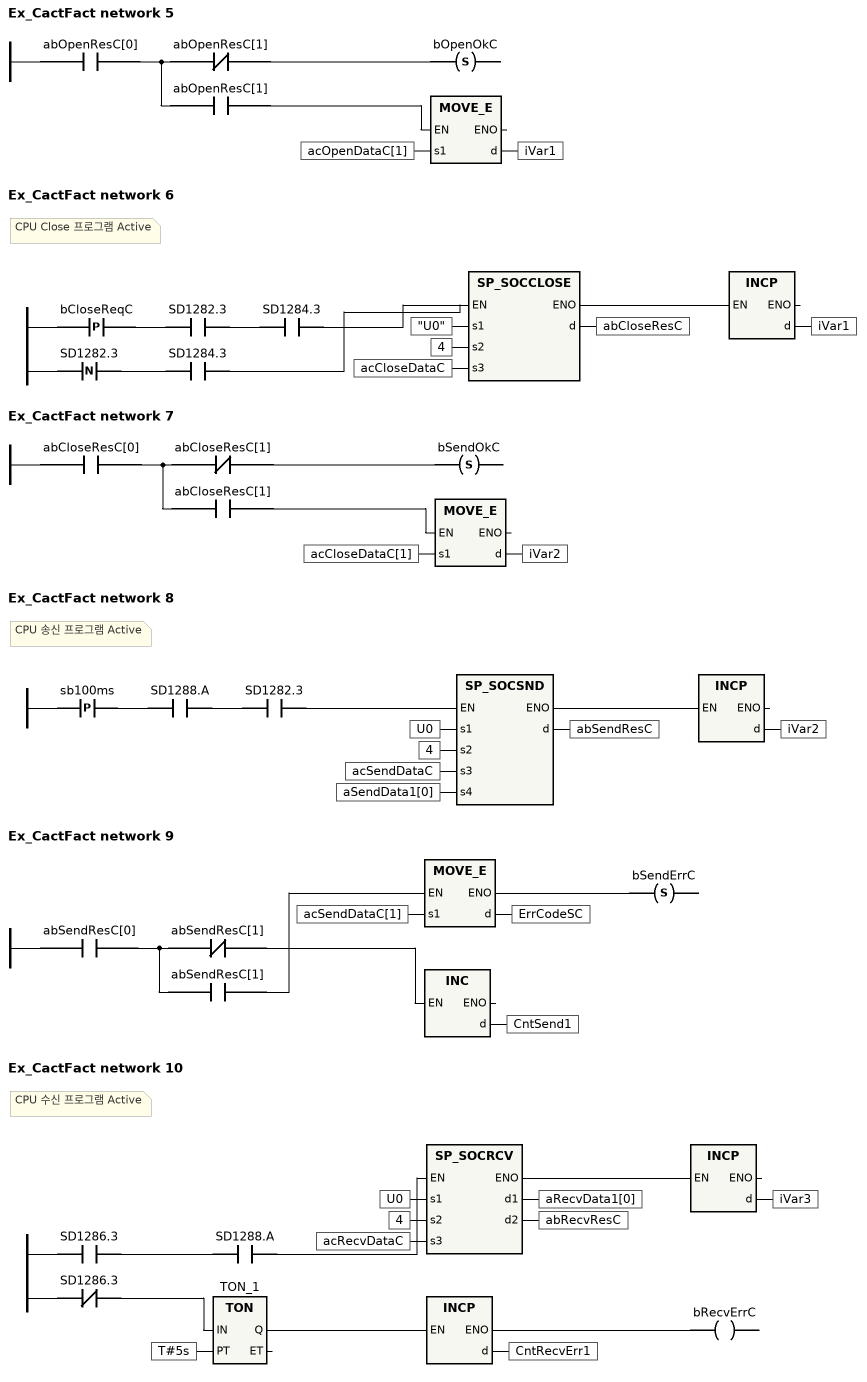
(* network 5 *)
SET(abOpenResC[0] AND NOT abOpenResC[1], bOpenOkC);
MOVE_E(abOpenResC[0] AND abOpenResC[1], acOpenDataC[1], iVar1);
(* network 6 *)
(* CPU Close 프로그램 Active *)
_e1 := SP_SOCCLOSE((LDP(TRUE, bCloseReqC) AND SD1282.3 AND SD1284.3) OR (LDF(TRUE, SD1282.3) AND SD1284.3), "U0", 4, acCloseDataC, abCloseResC);
INCP(_e1, iVar1);
(* network 7 *)
SET(abCloseResC[0] AND NOT abCloseResC[1], bSendOkC);
MOVE_E(abCloseResC[0] AND abCloseResC[1], acCloseDataC[1], iVar2);
(* network 8 *)
(* CPU 송신 프로그램 Active *)
_e1 := SP_SOCSND(LDP(TRUE, sb100ms) AND SD1288.A AND SD1282.3, U0, 4, acSendDataC, aSendData1[0], abSendResC);
INCP(_e1, iVar2);
(* network 9 *)
INC(abSendResC[0] AND NOT abSendResC[1], CntSend1);
_e1 := MOVE_E(abSendResC[0] AND abSendResC[1], acSendDataC[1], ErrCodeSC);
SET(_e1, bSendErrC);
(* network 10 *)
(* CPU 수신 프로그램 Active *)
_e1 := SP_SOCRCV(SD1286.3 AND SD1288.A, U0, 4, acRecvDataC, aRecvData1[0], abRecvResC);
INCP(_e1, iVar3);
TON_1(IN := NOT SD1286.3, PT := T#5s);
_e2 := INCP(TON_1.Q, CntRecvErr1);
bRecvErrC := _e2;
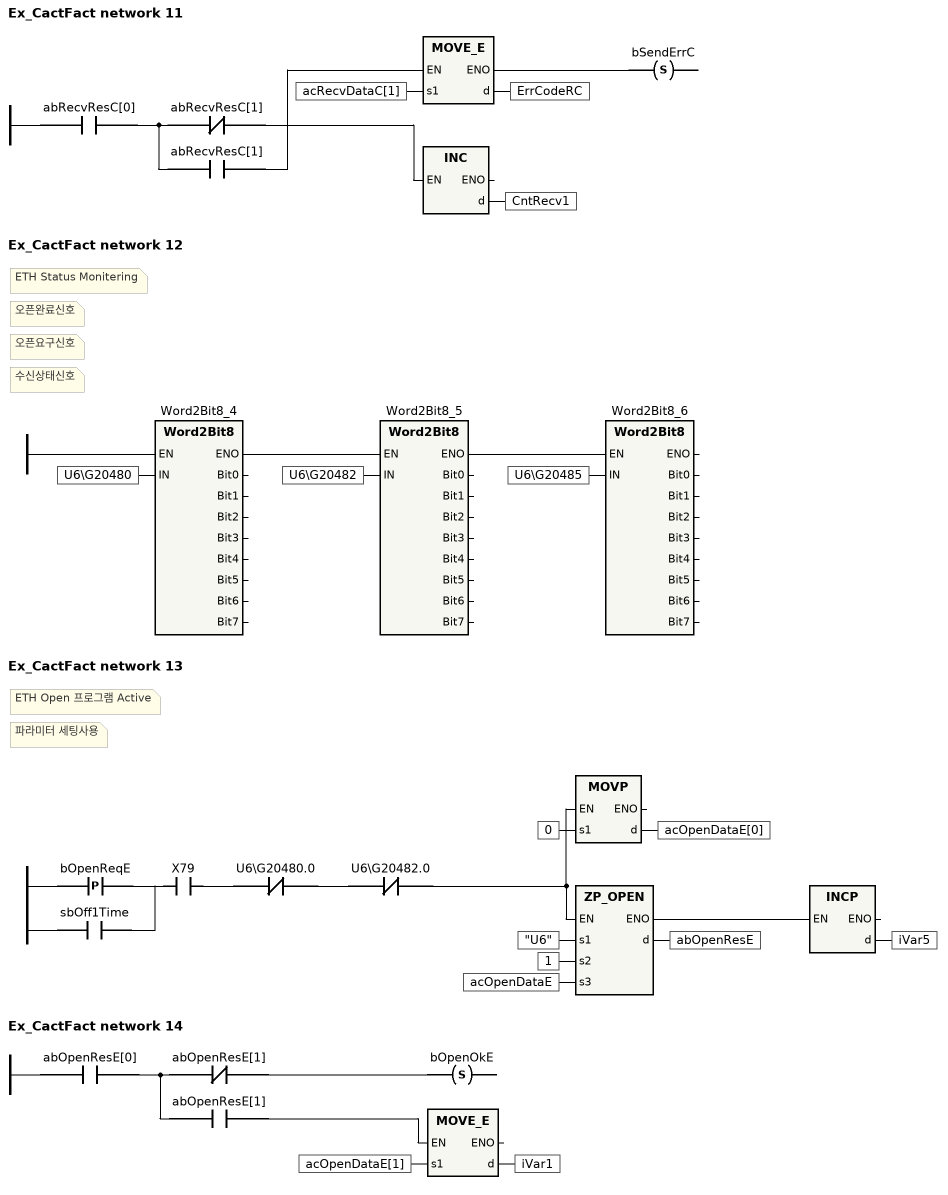
(* network 11 *)
INC(abRecvResC[0] AND NOT abRecvResC[1], CntRecv1);
_e1 := MOVE_E(abRecvResC[0] AND abRecvResC[1], acRecvDataC[1], ErrCodeRC);
SET(_e1, bSendErrC);
(* network 12 *)
(* ETH Status Monitering *)
(* 오픈완료신호 *)
(* 오픈요구신호 *)
(* 수신상태신호 *)
Word2Bit8_4(EN := TRUE, IN := U6\G20480);
Word2Bit8_5(EN := Word2Bit8_4.ENO, IN := U6\G20482);
Word2Bit8_6(EN := Word2Bit8_5.ENO, IN := U6\G20485);
(* network 13 *)
(* ETH Open 프로그램 Active *)
(* 파라미터 세팅사용 *)
_p1 := (((LDP(TRUE, bOpenReqE) OR sbOff1Time) AND X79) AND NOT U6\G20480.0) AND NOT U6\G20482.0;
MOVP(_p1, 0, acOpenDataE[0]);
_e2 := ZP_OPEN(_p1, "U6", 1, acOpenDataE, abOpenResE);
INCP(_e2, iVar5);
(* network 14 *)
SET(abOpenResE[0] AND NOT abOpenResE[1], bOpenOkE);
MOVE_E(abOpenResE[0] AND abOpenResE[1], acOpenDataE[1], iVar1);
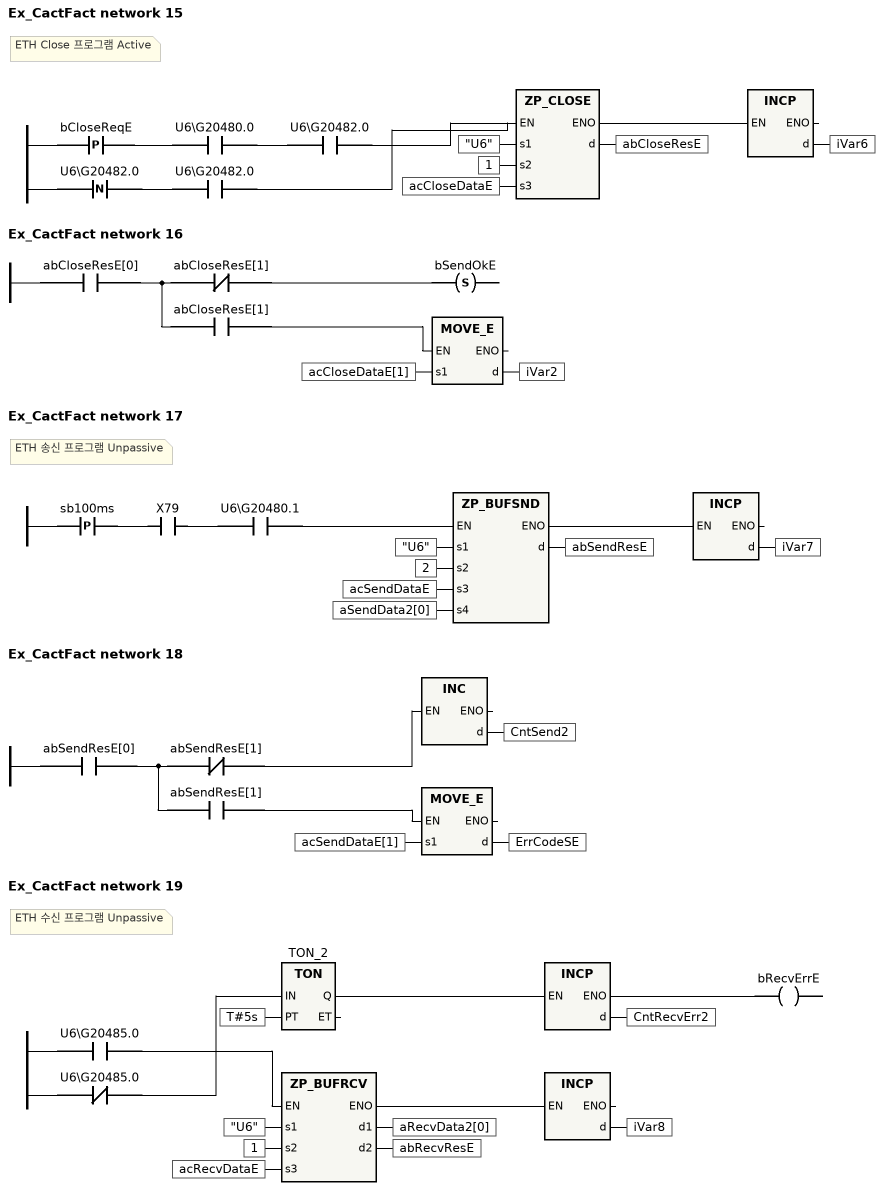
(* network 15 *)
(* ETH Close 프로그램 Active *)
_e1 := ZP_CLOSE((LDP(TRUE, bCloseReqE) AND U6\G20480.0 AND U6\G20482.0) OR (LDF(TRUE, U6\G20482.0) AND U6\G20482.0), "U6", 1, acCloseDataE, abCloseResE);
INCP(_e1, iVar6);
(* network 16 *)
SET(abCloseResE[0] AND NOT abCloseResE[1], bSendOkE);
MOVE_E(abCloseResE[0] AND abCloseResE[1], acCloseDataE[1], iVar2);
(* network 17 *)
(* ETH 송신 프로그램 Unpassive *)
_e1 := ZP_BUFSND(LDP(TRUE, sb100ms) AND X79 AND U6\G20480.1, "U6", 2, acSendDataE, aSendData2[0], abSendResE);
INCP(_e1, iVar7);
(* network 18 *)
INC(abSendResE[0] AND NOT abSendResE[1], CntSend2);
MOVE_E(abSendResE[0] AND abSendResE[1], acSendDataE[1], ErrCodeSE);
(* network 19 *)
(* ETH 수신 프로그램 Unpassive *)
_e1 := ZP_BUFRCV(U6\G20485.0, "U6", 1, acRecvDataE, aRecvData2[0], abRecvResE);
INCP(_e1, iVar8);
TON_2(IN := NOT U6\G20485.0, PT := T#5s);
_e2 := INCP(TON_2.Q, CntRecvErr2);
bRecvErrE := _e2;
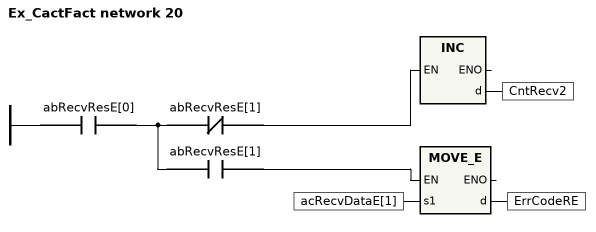
(* network 20 *)
INC(abRecvResE[0] AND NOT abRecvResE[1], CntRecv2);
MOVE_E(abRecvResE[0] AND abRecvResE[1], acRecvDataE[1], ErrCodeRE);
END_PROGRAM

PROGRAM Ex_CudpEudp
VAR
  bOpenReqC : BOOL;
  bCsetReq : BOOL;
  bOpenReqE : BOOL;
  bOpenOkC : BOOL;
  bOpenOkE : BOOL;
  bOpenErrC : BOOL;
  bOpenErrE : BOOL;
  abOpenResC : ARRAY [0..1] OF BOOL;
  abOpenResE : ARRAY [0..1] OF BOOL;
  acOpenDataC : ARRAY [0..9] OF INT;
  acCsetData : ARRAY [0..4] OF INT;
  acRdCtrl : ARRAY [0..9] OF INT;
  bSendReqC : BOOL;
  bSendReqE : BOOL;
  bSendOkC : BOOL;
  bSendOkE : BOOL;
  bSendErrC : BOOL;
  bSendErrE : BOOL;
  abSendResC : ARRAY [0..1] OF BOOL;
  abSendResE : ARRAY [0..1] OF BOOL;
  abSendResF : ARRAY [0..1] OF BOOL;
  acSendDataC : ARRAY [0..1] OF INT;
  acSendDataE : ARRAY [0..1] OF INT;
  acSendDataF : ARRAY [0..1] OF INT;
  bRecvOkC : BOOL;
  bRecvOkE : BOOL;
  bRecvOkF : BOOL;
  bRecvErrC : BOOL;
  bRecvErrE : BOOL;
  bRecvErrF : BOOL;
  abRecvResC : ARRAY [0..1] OF BOOL;
  abRecvRes3 : ARRAY [0..1] OF BOOL;
  abRecvRes13 : ARRAY [0..1] OF BOOL;
  acRecvDataC : ARRAY [0..1] OF INT;
  acRecvData3 : ARRAY [0..1] OF INT;
  acRecvData13 : ARRAY [0..1] OF INT;
  bCloseReqC : BOOL;
  bCloseOkC : BOOL;
  bCloseOkE : BOOL;
  bCloseErrC : BOOL;
  bCloseErrE : BOOL;
  abCloseResC : ARRAY [0..1] OF BOOL;
  abCloseResE : ARRAY [0..1] OF BOOL;
  acCloseDataC : ARRAY [0..1] OF INT;
  CntSend1 : INT;
  CntSend2 : INT;
  CntSend3 : INT;
  CntRecv1 : INT;
  CntRecvErr1 : INT;
  CntRecv2 : INT;
  CntRecv3 : INT;
  CntRecvErr2 : INT;
  CntRecvErr3 : INT;
  ErrCodeSC : INT;
  ErrCodeSE : INT;
  ErrCodeSF : INT;
  ErrCodeRC : INT;
  ErrCodeR3 : INT;
  ErrCodeR13 : INT;
  Mov4INT_1 : Mov4INT;
  Mov8INT_1 : Mov8INT;
  Mov4INT_2 : Mov4INT;
  Mov4INT_3 : Mov4INT;
  Mov4INT_4 : Mov4INT;
  Word2Bit8_1 : Word2Bit8;
  Word2Bit8_2 : Word2Bit8;
  Word2Bit8_3 : Word2Bit8;
  Word2Bit8_4 : Word2Bit8;
  Word2Bit8_5 : Word2Bit8;
  Word2Bit8_6 : Word2Bit8;
  TON_1 : TON;
  TON_2 : TON;
  TON_3 : TON;
  bCloseReqE : BOOL;
  acOpenDataE : ARRAY [0..9] OF INT;
  acCloseDataE : ARRAY [0..1] OF INT;
  ErrCodeOC : INT;
  ErrCodeOE : INT;
  ErrCodeCC : INT;
  ErrCodeCE : INT;
  bDelay : BOOL;
  bLedOff : BOOL;
  bChgReq : BOOL;
  bChgConn : BOOL;
  ChgPort : INT;
  CntRecv13 : INT;
  TON_13 : TON;
END_VAR
(* structured ladder/FBD written out as ST: instructions are called as NAME(EN, inputs, outputs); _pN, _eN, _tN stand for wires *)
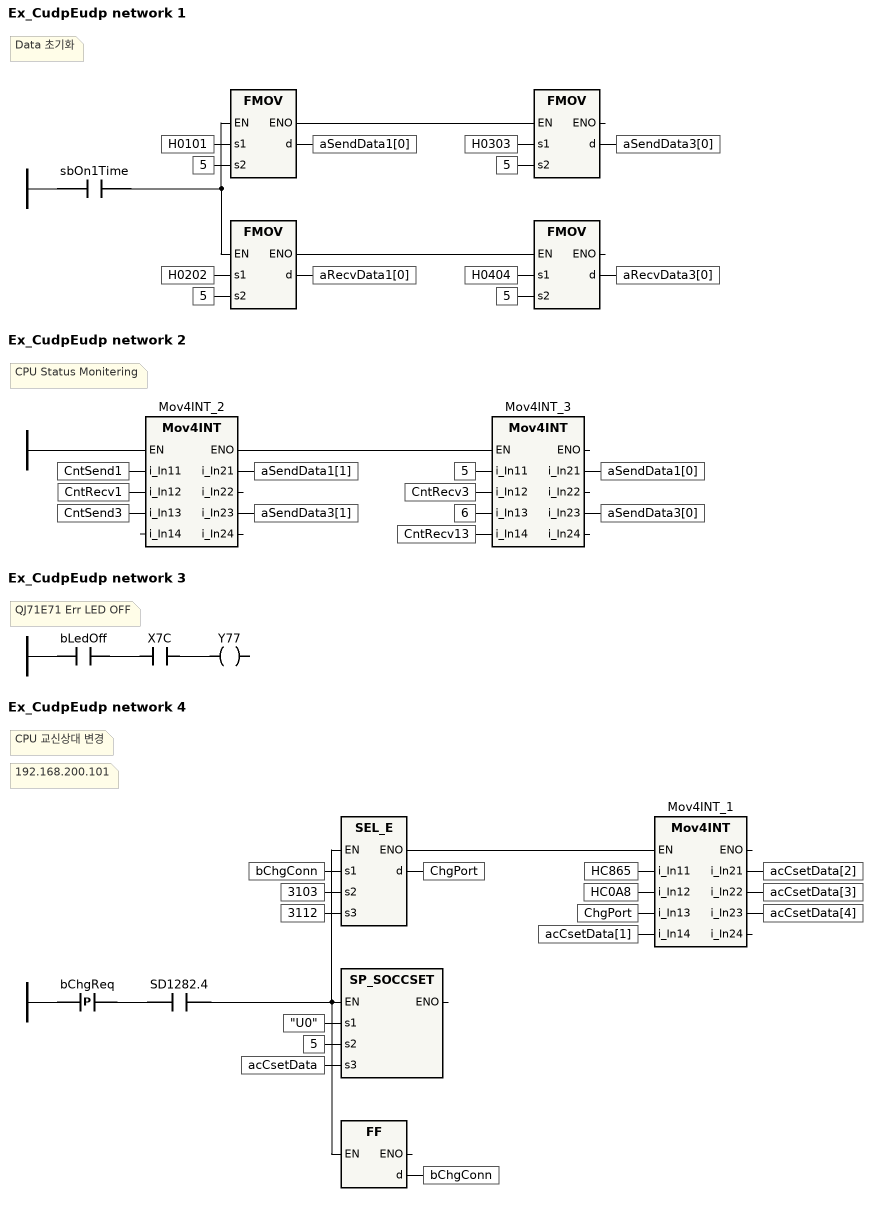
(* network 1 *)
(* Data 초기화 *)
_e1 := FMOV(sbOn1Time, H0101, 5, aSendData1[0]);
FMOV(_e1, H0303, 5, aSendData3[0]);
_e2 := FMOV(sbOn1Time, H0202, 5, aRecvData1[0]);
FMOV(_e2, H0404, 5, aRecvData3[0]);
(* network 2 *)
(* CPU Status Monitering *)
Mov4INT_2(EN := TRUE, i_In11 := CntSend1, i_In12 := CntRecv1, i_In13 := CntSend3, i_In21 => aSendData1[1], i_In23 => aSendData3[1]);
Mov4INT_3(EN := Mov4INT_2.ENO, i_In11 := 5, i_In12 := CntRecv3, i_In13 := 6, i_In14 := CntRecv13, i_In21 => aSendData1[0], i_In23 => aSendData3[0]);
(* network 3 *)
(* QJ71E71 Err LED OFF *)
Y77 := bLedOff AND X7C;
(* network 4 *)
(* CPU 교신상대 변경 *)
(* 192.168.200.101 *)
_p1 := LDP(TRUE, bChgReq) AND SD1282.4;
_e2 := SEL_E(_p1, bChgConn, 3103, 3112, ChgPort);
Mov4INT_1(EN := _e2, i_In11 := HC865, i_In12 := HC0A8, i_In13 := ChgPort, i_In14 := acCsetData[1], i_In21 => acCsetData[2], i_In22 => acCsetData[3], i_In23 => acCsetData[4]);
SP_SOCCSET(_p1, "U0", 5, acCsetData);
FF(_p1, bChgConn);
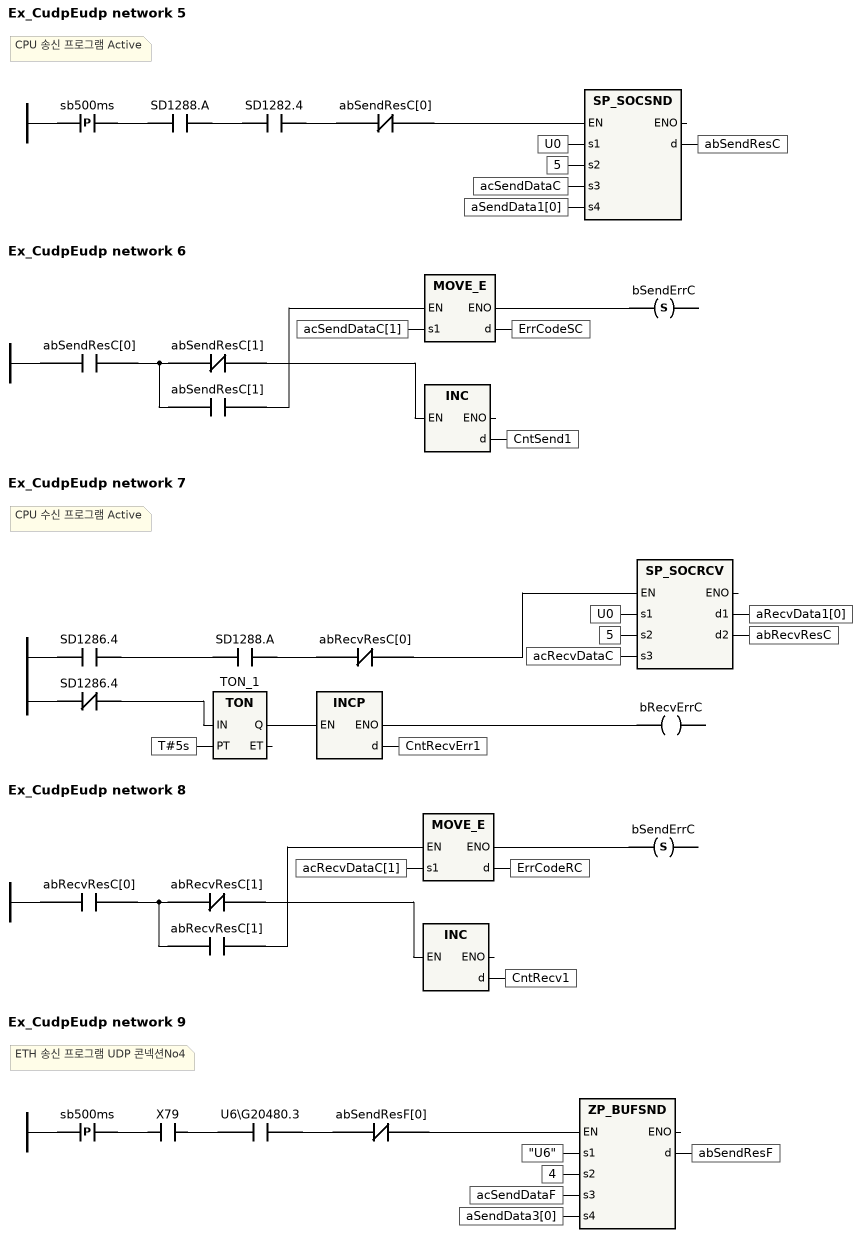
(* network 5 *)
(* CPU 송신 프로그램 Active *)
SP_SOCSND(LDP(TRUE, sb500ms) AND SD1288.A AND SD1282.4 AND NOT abSendResC[0], U0, 5, acSendDataC, aSendData1[0], abSendResC);
(* network 6 *)
INC(abSendResC[0] AND NOT abSendResC[1], CntSend1);
_e1 := MOVE_E(abSendResC[0] AND abSendResC[1], acSendDataC[1], ErrCodeSC);
SET(_e1, bSendErrC);
(* network 7 *)
(* CPU 수신 프로그램 Active *)
SP_SOCRCV(SD1286.4 AND SD1288.A AND NOT abRecvResC[0], U0, 5, acRecvDataC, aRecvData1[0], abRecvResC);
TON_1(IN := NOT SD1286.4, PT := T#5s);
_e1 := INCP(TON_1.Q, CntRecvErr1);
bRecvErrC := _e1;
(* network 8 *)
INC(abRecvResC[0] AND NOT abRecvResC[1], CntRecv1);
_e1 := MOVE_E(abRecvResC[0] AND abRecvResC[1], acRecvDataC[1], ErrCodeRC);
SET(_e1, bSendErrC);
(* network 9 *)
(* ETH 송신 프로그램 UDP 콘넥션No4 *)
ZP_BUFSND(LDP(TRUE, sb500ms) AND X79 AND U6\G20480.3 AND NOT abSendResF[0], "U6", 4, acSendDataF, aSendData3[0], abSendResF);
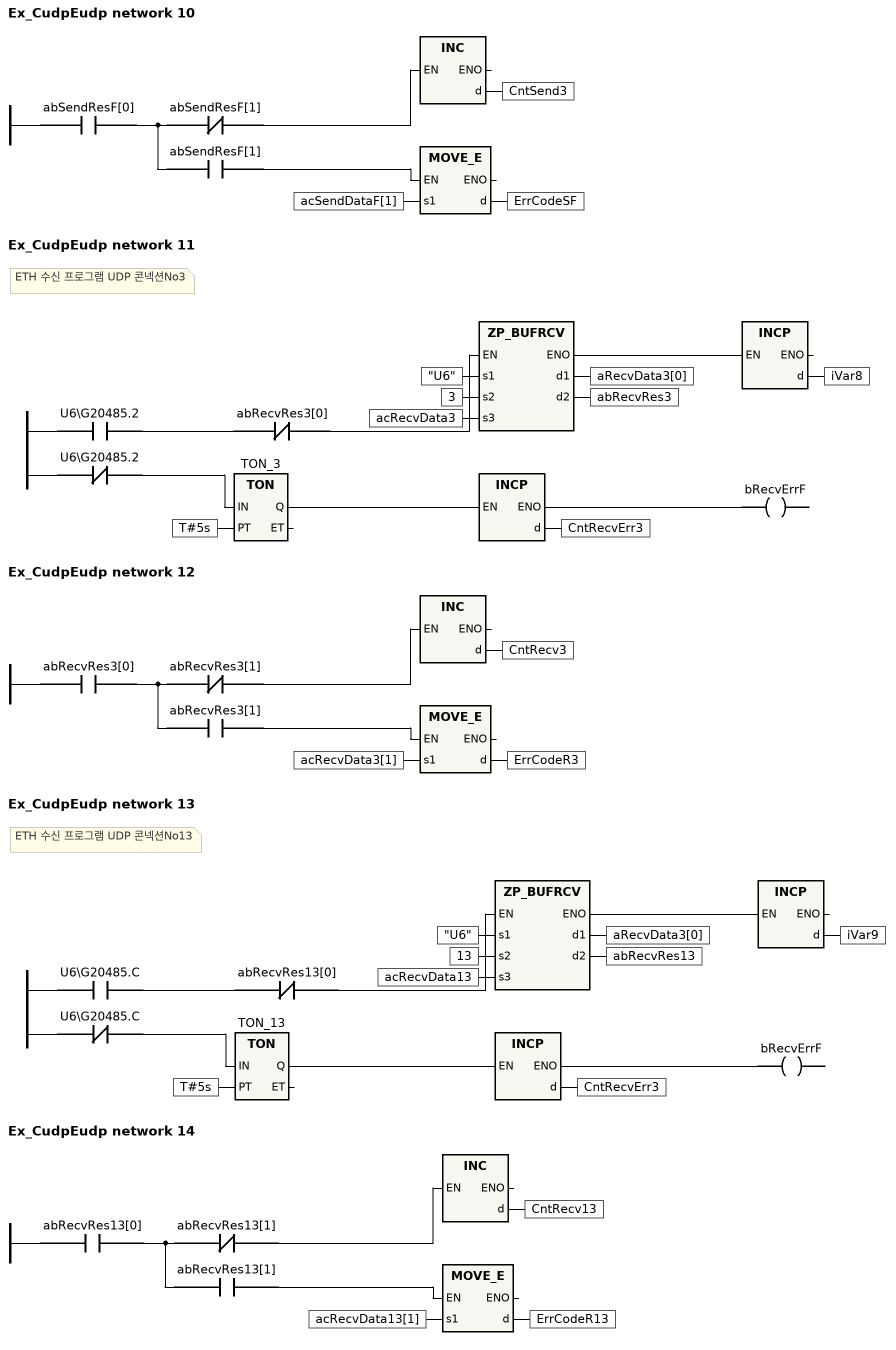
(* network 10 *)
INC(abSendResF[0] AND NOT abSendResF[1], CntSend3);
MOVE_E(abSendResF[0] AND abSendResF[1], acSendDataF[1], ErrCodeSF);
(* network 11 *)
(* ETH 수신 프로그램 UDP 콘넥션No3 *)
_e1 := ZP_BUFRCV(U6\G20485.2 AND NOT abRecvRes3[0], "U6", 3, acRecvData3, aRecvData3[0], abRecvRes3);
INCP(_e1, iVar8);
TON_3(IN := NOT U6\G20485.2, PT := T#5s);
_e2 := INCP(TON_3.Q, CntRecvErr3);
bRecvErrF := _e2;
(* network 12 *)
INC(abRecvRes3[0] AND NOT abRecvRes3[1], CntRecv3);
MOVE_E(abRecvRes3[0] AND abRecvRes3[1], acRecvData3[1], ErrCodeR3);
(* network 13 *)
(* ETH 수신 프로그램 UDP 콘넥션No13 *)
_e1 := ZP_BUFRCV(U6\G20485.C AND NOT abRecvRes13[0], "U6", 13, acRecvData13, aRecvData3[0], abRecvRes13);
INCP(_e1, iVar9);
TON_13(IN := NOT U6\G20485.C, PT := T#5s);
_e2 := INCP(TON_13.Q, CntRecvErr3);
bRecvErrF := _e2;
(* network 14 *)
INC(abRecvRes13[0] AND NOT abRecvRes13[1], CntRecv13);
MOVE_E(abRecvRes13[0] AND abRecvRes13[1], acRecvData13[1], ErrCodeR13);
END_PROGRAM

FUNCTION_BLOCK Word2Bit16
VAR_INPUT
  bEN : BOOL;
END_VAR
VAR_OUTPUT
  Bit0 : BOOL;
  Bit1 : BOOL;
  Bit2 : BOOL;
  Bit3 : BOOL;
  Bit4 : BOOL;
  Bit5 : BOOL;
  Bit6 : BOOL;
  Bit7 : BOOL;
  Bit8 : BOOL;
  Bit9 : BOOL;
  Bit10 : BOOL;
  Bit11 : BOOL;
  Bit12 : BOOL;
  Bit13 : BOOL;
  Bit14 : BOOL;
  Bit15 : BOOL;
END_VAR
VAR_INPUT
  InWord : WORD;
END_VAR
VAR_OUTPUT
  bENO : BOOL;
END_VAR
VAR
  InVal : WORD;
END_VAR
 
bENO := bEN;
InVal :=InWord;
Bit0 := (InVal AND 16#0001) = H0001;
Bit1 := (InVal AND 16#0002) = H0002;
Bit2 := (InVal AND 16#0004) = H0004;
Bit3 := (InVal AND 16#0008) = H0008;
Bit4 := (InVal AND 16#0010) = H0010;
Bit5 := (InVal AND 16#0020) = H0020;
Bit6 := (InVal AND 16#0040) = H0040;
Bit7 := (InVal AND 16#0080) = H0080;
Bit8 := (InVal AND 16#0100) = H0100;
Bit9 := (InVal AND 16#0200) = H0200;
Bit10 := (InVal AND 16#0400) = H0400;
Bit11 := (InVal AND 16#0800) = H0800;
Bit12 := (InVal AND 16#1000) = H1000;
Bit13 := (InVal AND 16#2000) = H2000;
Bit14 := (InVal AND 16#4000) = H4000;
Bit15 := (InVal AND 16#8000) = H8000;

(*
Bit0 := WORD_TO_BOOL(IN AND 16#0001);
Bit1 := WORD_TO_BOOL(SHR(IN AND 16#0002 , 1));
Bit2 := WORD_TO_BOOL(SHR(IN AND 16#0004 , 2));
Bit3 := WORD_TO_BOOL(SHR(IN AND 16#0008 , 3));
Bit4 := WORD_TO_BOOL(SHR(IN AND 16#0010 , 4));
Bit5 := WORD_TO_BOOL(SHR(IN AND 16#0020 , 5));
Bit6 := WORD_TO_BOOL(SHR(IN AND 16#0040 , 6));
Bit7 := WORD_TO_BOOL(SHR(IN AND 16#0080 , 7));
 
Bit8 := WORD_TO_BOOL(SHR(IN AND 16#0100 , 8));
Bit9 := WORD_TO_BOOL(SHR(IN AND 16#0200 , 9));
Bit10 := WORD_TO_BOOL(SHR(IN AND 16#0400 , 10));
Bit11 := WORD_TO_BOOL(SHR(IN AND 16#0800 , 11));
Bit12 := WORD_TO_BOOL(SHR(IN AND 16#1000 , 12));
Bit13 := WORD_TO_BOOL(SHR(IN AND 16#2000 , 13));
Bit14 := WORD_TO_BOOL(SHR(IN AND 16#4000 , 14));
Bit15 := WORD_TO_BOOL(SHR(IN AND 16#8000 , 15));
*)
END_FUNCTION_BLOCK

PROGRAM Ex_CpasEact
VAR
  bOpenReqC : BOOL;
  bCsetReq : BOOL;
  bOpenReqE : BOOL;
  bOpenOkC : BOOL;
  bOpenOkE : BOOL;
  bOpenErrC : BOOL;
  bOpenErrE : BOOL;
  abOpenResC : ARRAY [0..1] OF BOOL;
  abOpenResE : ARRAY [0..1] OF BOOL;
  acOpenDataC : ARRAY [0..9] OF INT;
  acCsetData : ARRAY [0..4] OF INT;
  acRdCtrl : ARRAY [0..9] OF INT;
  bSendReqC : BOOL;
  bSendReqE : BOOL;
  bSendOkC : BOOL;
  bSendOkE : BOOL;
  bSendErrC : BOOL;
  bSendErrE : BOOL;
  abSendResC : ARRAY [0..1] OF BOOL;
  abSendResE : ARRAY [0..1] OF BOOL;
  abSendResF : ARRAY [0..1] OF BOOL;
  acSendDataC : ARRAY [0..1] OF INT;
  acSendDataE : ARRAY [0..1] OF INT;
  acSendDataF : ARRAY [0..1] OF INT;
  bRecvOkC : BOOL;
  bRecvOkE : BOOL;
  bRecvOkF : BOOL;
  bRecvErrC : BOOL;
  bRecvErrE : BOOL;
  bRecvErrF : BOOL;
  abRecvResC : ARRAY [0..1] OF BOOL;
  abRecvResE : ARRAY [0..1] OF BOOL;
  abRecvResF : ARRAY [0..1] OF BOOL;
  acRecvDataC : ARRAY [0..1] OF INT;
  acRecvDataE : ARRAY [0..1] OF INT;
  acRecvDataF : ARRAY [0..1] OF INT;
  bCloseReqC : BOOL;
  bCloseOkC : BOOL;
  bCloseOkE : BOOL;
  bCloseErrC : BOOL;
  bCloseErrE : BOOL;
  abCloseResC : ARRAY [0..1] OF BOOL;
  abCloseResE : ARRAY [0..1] OF BOOL;
  acCloseDataC : ARRAY [0..1] OF INT;
  CntSend1 : INT;
  CntSend2 : INT;
  CntSend3 : INT;
  CntRecv1 : INT;
  CntRecvErr1 : INT;
  CntRecv2 : INT;
  CntRecv3 : INT;
  CntRecvErr2 : INT;
  CntRecvErr3 : INT;
  ErrCodeCC : INT;
  ErrCodeSE : INT;
  ErrCodeSF : INT;
  ErrCodeRC : INT;
  ErrCodeRE : INT;
  ErrCodeRF : INT;
  Mov4INT_1 : Mov4INT;
  Mov8INT_1 : Mov8INT;
  Mov4INT_2 : Mov4INT;
  Mov4INT_3 : Mov4INT;
  Mov4INT_4 : Mov4INT;
  Word2Bit8_1 : Word2Bit8;
  Word2Bit8_2 : Word2Bit8;
  Word2Bit8_3 : Word2Bit8;
  Word2Bit8_4 : Word2Bit8;
  Word2Bit8_5 : Word2Bit8;
  Word2Bit8_6 : Word2Bit8;
  TON_1 : TON;
  TON_2 : TON;
  TON_3 : TON;
  Status1 : WORD;
  Status2 : WORD;
  Status3 : WORD;
  Word2Bit16_1 : Word2Bit16;
  Word2Bit16_2 : Word2Bit16;
  Word2Bit16_3 : Word2Bit16;
  acOpenDataE : ARRAY [0..9] OF INT;
  acCloseDataE : ARRAY [0..1] OF INT;
  ErrCodeOE : INT;
  ErrCodeSC : INT;
  ErrCodeCE : INT;
  ErrCodeOC : INT;
  bCloseReqE : BOOL;
END_VAR
(* structured ladder/FBD written out as ST: instructions are called as NAME(EN, inputs, outputs); _pN, _eN, _tN stand for wires *)
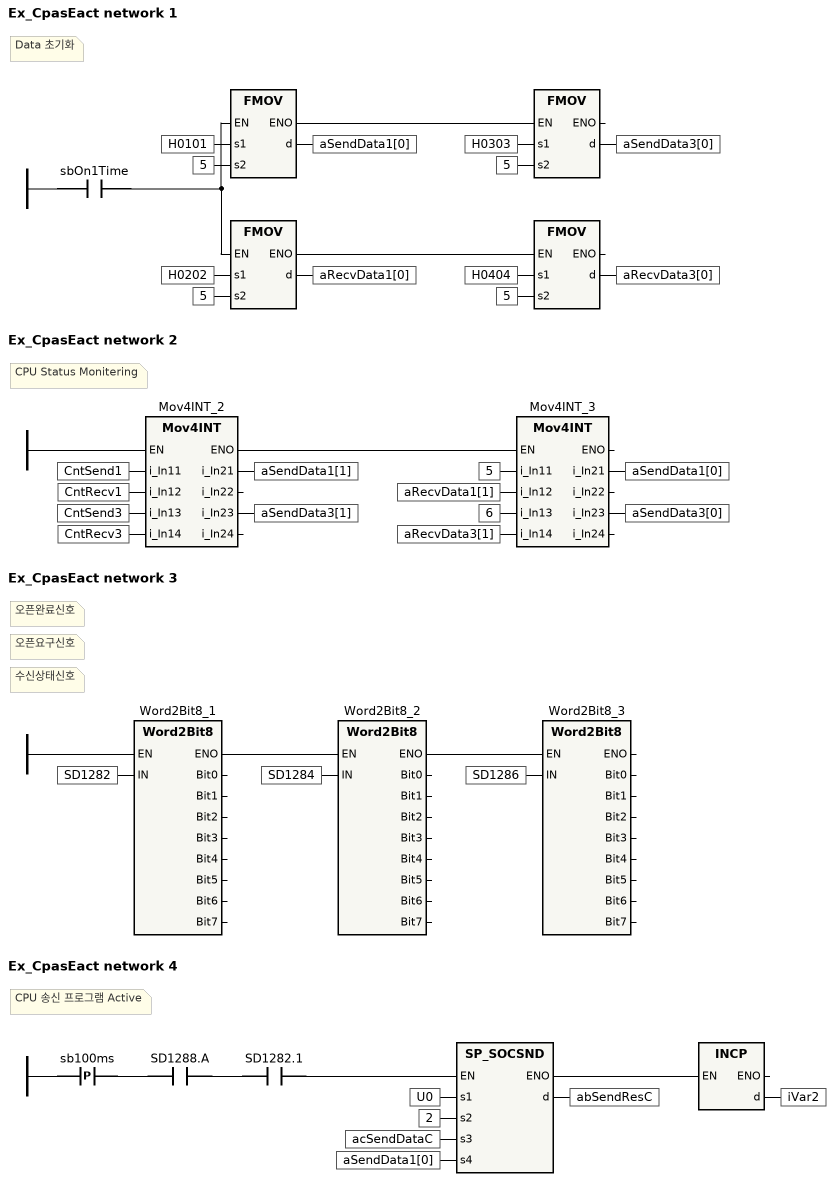
(* network 1 *)
(* Data 초기화 *)
_e1 := FMOV(sbOn1Time, H0101, 5, aSendData1[0]);
FMOV(_e1, H0303, 5, aSendData3[0]);
_e2 := FMOV(sbOn1Time, H0202, 5, aRecvData1[0]);
FMOV(_e2, H0404, 5, aRecvData3[0]);
(* network 2 *)
(* CPU Status Monitering *)
Mov4INT_2(EN := TRUE, i_In11 := CntSend1, i_In12 := CntRecv1, i_In13 := CntSend3, i_In14 := CntRecv3, i_In21 => aSendData1[1], i_In23 => aSendData3[1]);
Mov4INT_3(EN := Mov4INT_2.ENO, i_In11 := 5, i_In12 := aRecvData1[1], i_In13 := 6, i_In14 := aRecvData3[1], i_In21 => aSendData1[0], i_In23 => aSendData3[0]);
(* network 3 *)
(* 오픈완료신호 *)
(* 오픈요구신호 *)
(* 수신상태신호 *)
Word2Bit8_1(EN := TRUE, IN := SD1282);
Word2Bit8_2(EN := Word2Bit8_1.ENO, IN := SD1284);
Word2Bit8_3(EN := Word2Bit8_2.ENO, IN := SD1286);
(* network 4 *)
(* CPU 송신 프로그램 Active *)
_e1 := SP_SOCSND(LDP(TRUE, sb100ms) AND SD1288.A AND SD1282.1, U0, 2, acSendDataC, aSendData1[0], abSendResC);
INCP(_e1, iVar2);
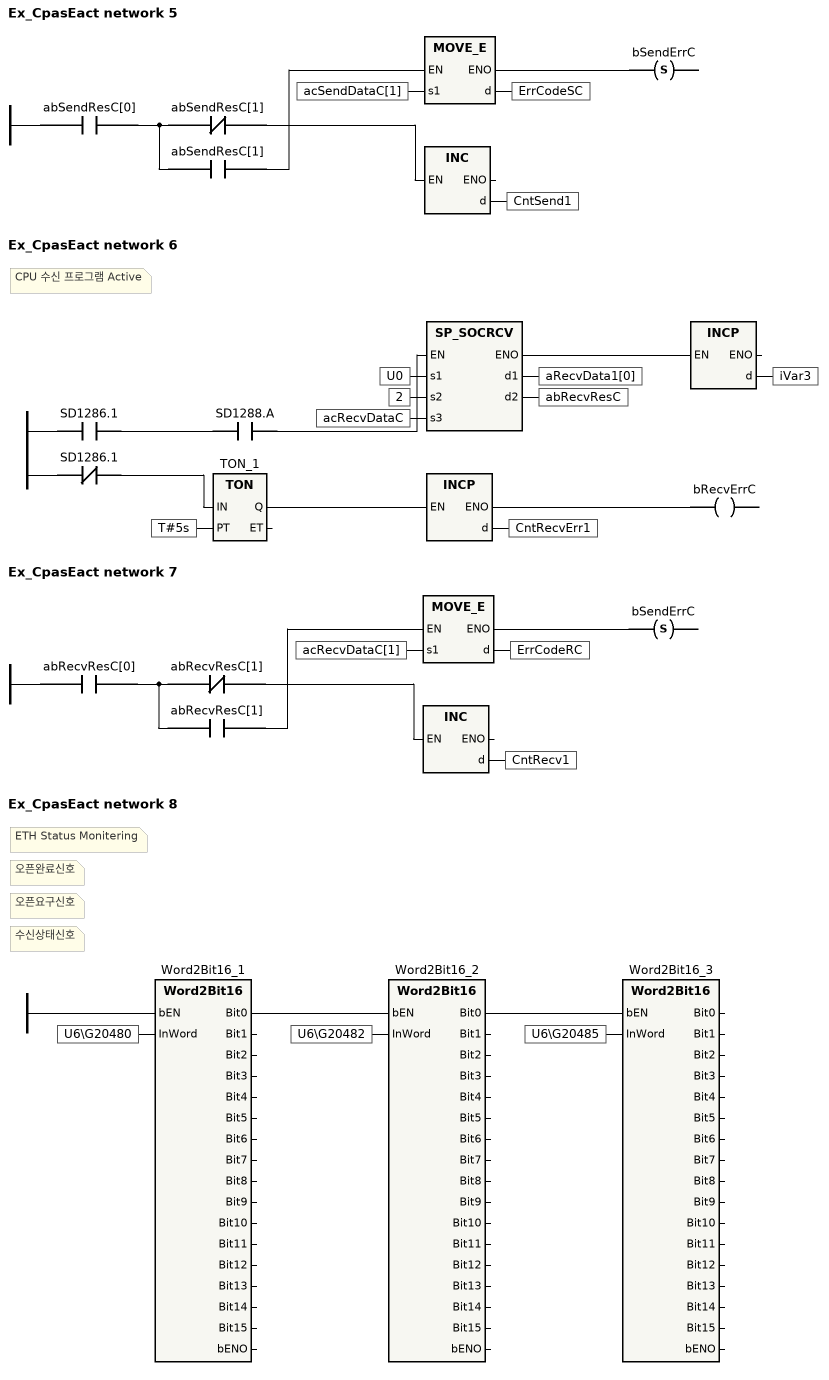
(* network 5 *)
INC(abSendResC[0] AND NOT abSendResC[1], CntSend1);
_e1 := MOVE_E(abSendResC[0] AND abSendResC[1], acSendDataC[1], ErrCodeSC);
SET(_e1, bSendErrC);
(* network 6 *)
(* CPU 수신 프로그램 Active *)
_e1 := SP_SOCRCV(SD1286.1 AND SD1288.A, U0, 2, acRecvDataC, aRecvData1[0], abRecvResC);
INCP(_e1, iVar3);
TON_1(IN := NOT SD1286.1, PT := T#5s);
_e2 := INCP(TON_1.Q, CntRecvErr1);
bRecvErrC := _e2;
(* network 7 *)
INC(abRecvResC[0] AND NOT abRecvResC[1], CntRecv1);
_e1 := MOVE_E(abRecvResC[0] AND abRecvResC[1], acRecvDataC[1], ErrCodeRC);
SET(_e1, bSendErrC);
(* network 8 *)
(* ETH Status Monitering *)
(* 오픈완료신호 *)
(* 오픈요구신호 *)
(* 수신상태신호 *)
Word2Bit16_1(bEN := TRUE, InWord := U6\G20480);
Word2Bit16_2(bEN := Word2Bit16_1.Bit0, InWord := U6\G20482);
Word2Bit16_3(bEN := Word2Bit16_2.Bit0, InWord := U6\G20485);
